FUNCTION_BLOCK "LAnyAxis_MC_OffsetRelative"   // FB30028, SCL
TITLE = LAnyAxis_MC_OffsetRelative
{ S7_Optimized_Access := 'TRUE' }
AUTHOR : tech.team.motioncontrol@siemens.com
FAMILY : AnyAxis
VERSION : 1.1
// Support: tech.team.motioncontrol@siemens.com 
// This block is for internal use only
   VAR_INPUT
      Slave : DB_ANY;   // See corresponding parameter of MC_ instruction in TIA Portal help (information system)
      Execute : Bool;   // See corresponding parameter of MC_ instruction in TIA Portal help (information system)
      Offset : LReal;   // See corresponding parameter of MC_ instruction in TIA Portal help (information system)
      ProfileReference : DInt := 1;   // See corresponding parameter of MC_ instruction in TIA Portal help (information system)
      OffsetDistance : LReal;   // See corresponding parameter of MC_ instruction in TIA Portal help (information system)
      StartPosition : LReal;   // See corresponding parameter of MC_ instruction in TIA Portal help (information system)
      Direction : DInt := 3;   // See corresponding parameter of MC_ instruction in TIA Portal help (information system)
   END_VAR
   VAR_OUTPUT
      Done : Bool;   // See corresponding parameter of MC_ instruction in TIA Portal help (information system)
      Busy : Bool;   // See corresponding parameter of MC_ instruction in TIA Portal help (information system)
      CommandAborted : Bool;   // See corresponding parameter of MC_ instruction in TIA Portal help (information system)
      Error : Bool;   // See corresponding parameter of MC_ instruction in TIA Portal help (information system)
      ErrorID : Word;   // See corresponding parameter of MC_ instruction in TIA Portal help (information system)
      CoveredOffset : LReal;   // See corresponding parameter of MC_ instruction in TIA Portal help (information system)
      StartOffset : Bool;   // See corresponding parameter of MC_ instruction in TIA Portal help (information system)
   END_VAR
   VAR CONSTANT
      ERROR_INVALID_TECHNOLOGY_OBJECT : Word := 16#8002;   // See corresponding parameter of MC_ instruction in TIA Portal help (information system)
   END_VAR
BEGIN
   REGION HEADER
     //================================================================================
     // SIEMENS AG
     // (c)Copyright 2021 All Rights Reserved
     //--------------------------------------------------------------------------------
     // Library: LAnyAxis 
     // Tested with: S7-1515-2 PN
     // Engineering: TIA Portal V17
     // Restrictions: -
     // Requirements: S7-1500 FW 2.9 
     // Functionality: Conversion DB_ANY --> TO_Axis
     // Support: tech.team.motioncontrol@siemens.com
     // Note: Parameter comments are only available in language 'English (United States)'
     //--------------------------------------------------------------------------------
     // Change log table:
     // Version  Date        Expert in charge  Changes applied
     // 01.00.00 10.03.2020  RS                First released version
     // 01.01.00 24.02.2021  RS                Update MC V6.0
     //================================================================================
   END_REGION

   #Done := FALSE;
   #Busy := FALSE;
   #CommandAborted := FALSE;
   #CoveredOffset := 0.0;
   #StartOffset := FALSE;

   IF #Execute THEN
     #Error := TRUE;
     #ErrorID := #ERROR_INVALID_TECHNOLOGY_OBJECT;
   ELSE
     #Error := FALSE;
     #ErrorID := 16#0000;
   END_IF;
END_FUNCTION_BLOCK

FUNCTION_BLOCK "LAnyAxis_MC_OffsetAbsolute"   // FB30029, SCL
TITLE = LAnyAxis_MC_OffsetAbsolute
{ S7_Optimized_Access := 'TRUE' }
AUTHOR : tech.team.motioncontrol@siemens.com
FAMILY : AnyAxis
VERSION : 1.1
// Support: tech.team.motioncontrol@siemens.com 
// This block is for internal use only
   VAR_INPUT
      Slave : DB_ANY;   // See corresponding parameter of MC_ instruction in TIA Portal help (information system)
      Execute : Bool;   // See corresponding parameter of MC_ instruction in TIA Portal help (information system)
      Offset : LReal;   // See corresponding parameter of MC_ instruction in TIA Portal help (information system)
      ProfileReference : DInt := 1;   // See corresponding parameter of MC_ instruction in TIA Portal help (information system)
      OffsetDistance : LReal;   // See corresponding parameter of MC_ instruction in TIA Portal help (information system)
      StartPosition : LReal;   // See corresponding parameter of MC_ instruction in TIA Portal help (information system)
      Direction : DInt := 3;   // See corresponding parameter of MC_ instruction in TIA Portal help (information system)
   END_VAR
   VAR_OUTPUT
      Done : Bool;   // See corresponding parameter of MC_ instruction in TIA Portal help (information system)
      Busy : Bool;   // See corresponding parameter of MC_ instruction in TIA Portal help (information system)
      CommandAborted : Bool;   // See corresponding parameter of MC_ instruction in TIA Portal help (information system)
      Error : Bool;   // See corresponding parameter of MC_ instruction in TIA Portal help (information system)
      ErrorID : Word;   // See corresponding parameter of MC_ instruction in TIA Portal help (information system)
      AbsoluteOffset : LReal;   // See corresponding parameter of MC_ instruction in TIA Portal help (information system)
      StartOffset : Bool;   // See corresponding parameter of MC_ instruction in TIA Portal help (information system)
   END_VAR
   VAR CONSTANT
      ERROR_INVALID_TECHNOLOGY_OBJECT : Word := 16#8002;   // See corresponding parameter of MC_ instruction in TIA Portal help (information system)
   END_VAR
BEGIN
   REGION HEADER
     //================================================================================
     // SIEMENS AG
     // (c)Copyright 2021 All Rights Reserved
     //--------------------------------------------------------------------------------
     // Library: LAnyAxis 
     // Tested with: S7-1515-2 PN
     // Engineering: TIA Portal V17
     // Restrictions: -
     // Requirements: S7-1500 FW 2.9 
     // Functionality: Conversion DB_ANY --> TO_Axis
     // Support: tech.team.motioncontrol@siemens.com
     // Note: Parameter comments are only available in language 'English (United States)'
     //--------------------------------------------------------------------------------
     // Change log table:
     // Version  Date        Expert in charge  Changes applied
     // 01.00.00 10.03.2020  RS                First released version
     // 01.01.00 24.02.2021  RS                Update MC V6.0
     //================================================================================
   END_REGION

   #Done := FALSE;
   #Busy := FALSE;
   #CommandAborted := FALSE;
   #AbsoluteOffset := 0.0;
   #StartOffset := FALSE;

   IF #Execute THEN
     #Error := TRUE;
     #ErrorID := #ERROR_INVALID_TECHNOLOGY_OBJECT;
   ELSE
     #Error := FALSE;
     #ErrorID := 16#0000;
   END_IF;
END_FUNCTION_BLOCK

FUNCTION_BLOCK "LAnyAxis_MC_GearOut"   // FB30032, SCL
TITLE = LAnyAxis_MC_GearOut
{ S7_Optimized_Access := 'TRUE' }
AUTHOR : tech.team.motioncontrol@siemens.com
FAMILY : AnyAxis
VERSION : 1.1
// Support: tech.team.motioncontrol@siemens.com 
// This block is for internal use only
   VAR_INPUT
      Slave : DB_ANY;   // See corresponding parameter of MC_ instruction in TIA Portal help (information system)
      Execute : Bool;   // See corresponding parameter of MC_ instruction in TIA Portal help (information system)
      SlavePosition : LReal;   // See corresponding parameter of MC_ instruction in TIA Portal help (information system)
      SyncProfileReference : DInt := 1;   // See corresponding parameter of MC_ instruction in TIA Portal help (information system)
      MasterStopDistance : LReal;   // See corresponding parameter of MC_ instruction in TIA Portal help (information system)
      Deceleration : LReal := -1.0;   // See corresponding parameter of MC_ instruction in TIA Portal help (information system)
      Jerk : LReal := -1.0;   // See corresponding parameter of MC_ instruction in TIA Portal help (information system)
      SyncOutDirection : DInt := 3;   // See corresponding parameter of MC_ instruction in TIA Portal help (information system)
   END_VAR
   VAR_OUTPUT
      StartSyncOut : Bool;   // See corresponding parameter of MC_ instruction in TIA Portal help (information system)
      Done : Bool;   // See corresponding parameter of MC_ instruction in TIA Portal help (information system)
      Busy : Bool;   // See corresponding parameter of MC_ instruction in TIA Portal help (information system)
      CommandAborted : Bool;   // See corresponding parameter of MC_ instruction in TIA Portal help (information system)
      Error : Bool;   // See corresponding parameter of MC_ instruction in TIA Portal help (information system)
      ErrorID : Word;   // See corresponding parameter of MC_ instruction in TIA Portal help (information system)
   END_VAR
   VAR CONSTANT
      ERROR_INVALID_TECHNOLOGY_OBJECT : Word := 16#8002;   // See corresponding parameter of MC_ instruction in TIA Portal help (information system)
   END_VAR
BEGIN
   REGION HEADER
     //================================================================================
     // SIEMENS AG
     // (c)Copyright 2021 All Rights Reserved
     //--------------------------------------------------------------------------------
     // Library: LAnyAxis 
     // Tested with: S7-1515-2 PN
     // Engineering: TIA Portal V17
     // Restrictions: -
     // Requirements: S7-1500 FW 2.9 
     // Functionality: Conversion DB_ANY --> TO_Axis
     // Support: tech.team.motioncontrol@siemens.com
     // Note: Parameter comments are only available in language 'English (United States)'
     //--------------------------------------------------------------------------------
     // Change log table:
     // Version  Date        Expert in charge  Changes applied
     // 01.00.00 10.03.2020  RS                First released version
     // 01.01.00 24.02.2021  RS                Update MC V6.0
     //================================================================================
   END_REGION

   #StartSyncOut := FALSE;
   #Done := FALSE;
   #Busy := FALSE;
   #CommandAborted := FALSE;

   IF #Execute THEN
     #Error := TRUE;
     #ErrorID := #ERROR_INVALID_TECHNOLOGY_OBJECT;
   ELSE
     #Error := FALSE;
     #ErrorID := 16#0000;
   END_IF;
END_FUNCTION_BLOCK

FUNCTION_BLOCK "LAnyAxis_MC_CamOut"   // FB30033, SCL
TITLE = LAnyAxis_MC_CamOut
{ S7_Optimized_Access := 'TRUE' }
AUTHOR : tech.team.motioncontrol@siemens.com
FAMILY : AnyAxis
VERSION : 1.1
// Support: tech.team.motioncontrol@siemens.com 
// This block is for internal use only
   VAR_INPUT
      Slave : DB_ANY;   // See corresponding parameter of MC_ instruction in TIA Portal help (information system)
      Execute : Bool;   // See corresponding parameter of MC_ instruction in TIA Portal help (information system)
      SlavePosition : LReal;   // See corresponding parameter of MC_ instruction in TIA Portal help (information system)
      SyncProfileReference : DInt := 1;   // See corresponding parameter of MC_ instruction in TIA Portal help (information system)
      MasterStopDistance : LReal;   // See corresponding parameter of MC_ instruction in TIA Portal help (information system)
      Deceleration : LReal := -1.0;   // See corresponding parameter of MC_ instruction in TIA Portal help (information system)
      Jerk : LReal := -1.0;   // See corresponding parameter of MC_ instruction in TIA Portal help (information system)
      SyncOutDirection : DInt := 3;   // See corresponding parameter of MC_ instruction in TIA Portal help (information system)
   END_VAR
   VAR_OUTPUT
      StartSyncOut : Bool;   // See corresponding parameter of MC_ instruction in TIA Portal help (information system)
      Done : Bool;   // See corresponding parameter of MC_ instruction in TIA Portal help (information system)
      Busy : Bool;   // See corresponding parameter of MC_ instruction in TIA Portal help (information system)
      CommandAborted : Bool;   // See corresponding parameter of MC_ instruction in TIA Portal help (information system)
      Error : Bool;   // See corresponding parameter of MC_ instruction in TIA Portal help (information system)
      ErrorID : Word;   // See corresponding parameter of MC_ instruction in TIA Portal help (information system)
   END_VAR
   VAR CONSTANT
      ERROR_INVALID_TECHNOLOGY_OBJECT : Word := 16#8002;   // See corresponding parameter of MC_ instruction in TIA Portal help (information system)
   END_VAR
BEGIN
   REGION HEADER
     //================================================================================
     // SIEMENS AG
     // (c)Copyright 2021 All Rights Reserved
     //--------------------------------------------------------------------------------
     // Library: LAnyAxis 
     // Tested with: S7-1515-2 PN
     // Engineering: TIA Portal V17
     // Restrictions: -
     // Requirements: S7-1500 FW 2.9 
     // Functionality: Conversion DB_ANY --> TO_Axis
     // Support: tech.team.motioncontrol@siemens.com
     // Note: Parameter comments are only available in language 'English (United States)'
     //--------------------------------------------------------------------------------
     // Change log table:
     // Version  Date        Expert in charge  Changes applied
     // 01.00.00 10.03.2020  RS                First released version
     // 01.01.00 24.02.2021  RS                Update MC V6.0
     //================================================================================
   END_REGION

   #StartSyncOut := FALSE;
   #Done := FALSE;
   #Busy := FALSE;
   #CommandAborted := FALSE;

   IF #Execute THEN
     #Error := TRUE;
     #ErrorID := #ERROR_INVALID_TECHNOLOGY_OBJECT;
   ELSE
     #Error := FALSE;
     #ErrorID := 16#0000;
   END_IF;
END_FUNCTION_BLOCK

// folder: LAnyAxis_Blocks/LAnyAxis_MC_SynchronousMotion/InternalSubBlocks/MC_GearIn

FUNCTION "LAnyAxis_UnpubGearInMasterExtEncoder" : Void   // FC30000, SCL
TITLE = LAnyAxis_UnpubGearInMasterExtEncoder
{ S7_Optimized_Access := 'TRUE' }
AUTHOR : tech.team.motioncontrol@siemens.com
FAMILY : AnyAxis
VERSION : 1.0
// Support: tech.team.motioncontrol@siemens.com
   VAR_INPUT
      slave : TO_SynchronousAxis;   // Slave axis specification
      master : TO_ExternalEncoder;   // Master axis specification
   END_VAR
   VAR_IN_OUT
      instMC : MC_GEARIN;   // Instance of MC_Instruction
   END_VAR
   // Ret_Val : No return value
BEGIN
   // Call of MC_Instruction
   #instMC(Master := #master,
           Slave := #slave);
END_FUNCTION

FUNCTION "LAnyAxis_UnpubGearInMasterPosAxis" : Void   // FC30001, SCL
TITLE = LAnyAxis_UnpubGearInMasterPosAxis
{ S7_Optimized_Access := 'TRUE' }
AUTHOR : tech.team.motioncontrol@siemens.com
FAMILY : AnyAxis
VERSION : 1.0
// Support: tech.team.motioncontrol@siemens.com
   VAR_INPUT
      slave : TO_SynchronousAxis;   // Slave axis specification
      master : TO_PositioningAxis;   // Master axis specification
   END_VAR
   VAR_IN_OUT
      instMC : MC_GEARIN;   // Instance of MC_Instruction
   END_VAR
   // Ret_Val : No return value
BEGIN
   // Call of MC_Instruction
   #instMC(Master := #master,
           Slave := #slave);
END_FUNCTION

FUNCTION "LAnyAxis_UnpubGearInMasterSyncAxis" : Void   // FC30002, SCL
TITLE = LAnyAxis_UnpubGearInMasterSyncAxis
{ S7_Optimized_Access := 'TRUE' }
AUTHOR : tech.team.motioncontrol@siemens.com
FAMILY : AnyAxis
VERSION : 1.0
// Support: tech.team.motioncontrol@siemens.com
   VAR_INPUT
      slave : TO_SynchronousAxis;   // Slave axis specification
      master : TO_SynchronousAxis;   // Master axis specification
   END_VAR
   VAR_IN_OUT
      instMC : MC_GEARIN;   // Instance of MC_Instruction
   END_VAR
   // Ret_Val : No return value
BEGIN
   // Call of MC_Instruction
   #instMC(Master := #master,
           Slave := #slave);
END_FUNCTION

// folder: LAnyAxis_Blocks/LAnyAxis_MC_TorqueData

FUNCTION_BLOCK "LAnyAxis_MC_TorqueLimiting"   // FB30042, SCL
TITLE = LAnyAxis_MC_TorqueLimiting
{ S7_Optimized_Access := 'TRUE' }
AUTHOR : tech.team.motioncontrol@siemens.com
FAMILY : AnyAxis
VERSION : 1.0
// Support: tech.team.motioncontrol@siemens.com 
// See corresponding MC_ instruction in TIA Portal help (information system)
   VAR_INPUT
      Axis : DB_ANY;   // See corresponding parameter of MC_ instruction in TIA Portal help (information system)
      Enable : Bool;   // See corresponding parameter of MC_ instruction in TIA Portal help (information system)
      Limit : LReal := -1.0;   // See corresponding parameter of MC_ instruction in TIA Portal help (information system)
      Mode : DInt;   // See corresponding parameter of MC_ instruction in TIA Portal help (information system)
   END_VAR
   VAR_OUTPUT
      InClamping : Bool;   // See corresponding parameter of MC_ instruction in TIA Portal help (information system)
      InLimitation : Bool;   // See corresponding parameter of MC_ instruction in TIA Portal help (information system)
      Busy : Bool;   // See corresponding parameter of MC_ instruction in TIA Portal help (information system)
      Error : Bool;   // See corresponding parameter of MC_ instruction in TIA Portal help (information system)
      ErrorId : Word;   // See corresponding parameter of MC_ instruction in TIA Portal help (information system)
   END_VAR
   VAR
      instMC : MC_TORQUELIMITING;   // Instance of MC_Instruction
      statEnableOld : Bool;   // Old value of execute
      statAxis : DB_ANY;   // Internal variable of axis
      statAxisType : Int;   // Actual state / axis type
   END_VAR
   VAR CONSTANT
      ERROR_INVALID_TECHNOLOGY_OBJECT : Word := 16#8002;   // See corresponding parameter of MC_ instruction in TIA Portal help (information system)
      IDLE : Int := 0;   // State idle
      INVALID_AXIS : Int := -1;   // Axis type: Invalid
      SPEED_AXIS : Int := 2;   // Axis type: Speed axis
      POSITIONING_AXIS : Int := 3;   // Axis type: Positioning axis
      SYNCHRONOUS_AXIS : Int := 4;   // Axis type: Synchronous axis
   END_VAR
BEGIN
   REGION HEADER
     //================================================================================
     // SIEMENS AG
     // (c)Copyright 2020 All Rights Reserved
     //--------------------------------------------------------------------------------
     // Library: LAnyAxis 
     // Tested with: S7-1515-2 PN
     // Engineering: TIA Portal V16
     // Restrictions: -
     // Requirements: S7-1500 FW 2.8.1
     // Functionality: Conversion DB_ANY --> TO_Axis
     // Support: tech.team.motioncontrol@siemens.com
     // Note: Parameter comments are only available in language 'English (United States)'
     //--------------------------------------------------------------------------------
     // Change log table:
     // Version  Date        Expert in charge  Changes applied
     // 01.00.00 10.03.2020  RS                First released version
     //================================================================================
   END_REGION

   REGION ENABLE
     IF (#statAxisType = #IDLE) AND #Enable THEN
       // Check axis type
       CASE TypeOfDB(#Axis) OF
         TO_POSITIONINGAXIS:
           #statAxisType := #POSITIONING_AXIS;
           #statAxis := #Axis;

         TO_SYNCHRONOUSAXIS:
           #statAxisType := #SYNCHRONOUS_AXIS;
           #statAxis := #Axis;

         TO_SPEEDAXIS:
           #statAxisType := #SPEED_AXIS;
           #statAxis := #Axis;

         ELSE
           #statAxisType := #INVALID_AXIS;
           #statAxis := 0;
       END_CASE;

     ELSIF NOT #Enable AND (#statAxisType = #INVALID_AXIS) THEN
       #statAxisType := #IDLE;

       // Outputs
       #InClamping := FALSE;
       #InLimitation := FALSE;
       #Busy := FALSE;
       #Error := FALSE;
       #ErrorId := 16#0;
     END_IF;

     // Edge detection
     #statEnableOld := #Enable;
   END_REGION

   CASE #statAxisType OF
     #IDLE:
       ;

     #POSITIONING_AXIS,
     #SYNCHRONOUS_AXIS,
     #SPEED_AXIS:
       REGION VALID_AXIS
         // Inputs
         #instMC.Enable := #Enable;
         #instMC.Limit := #Limit;
         #instMC.Mode := #Mode;

         // Call of MC instruction
         CASE #statAxisType OF
           #POSITIONING_AXIS:
             "LAnyAxis_UnpubTorqueLimitingPosAxis"(axis := #statAxis,
                                                   instMC := #instMC);
           #SYNCHRONOUS_AXIS:
             "LAnyAxis_UnpubTorqueLimitingSyncAxis"(axis := #statAxis,
                                                    instMC := #instMC);
           #SPEED_AXIS:
             #instMC(Axis := #statAxis);
         END_CASE;

         // Outputs
         #InClamping := #instMC.InClamping;
         #InLimitation := #instMC.InLimitation;
         #Busy := #instMC.Busy;
         #Error := #instMC.Error;
         #ErrorId := #instMC.ErrorId;

         // Status of MC instruction
         IF NOT #instMC.Busy
           AND NOT #instMC.Error
         THEN
           // Not active
           #statAxisType := #IDLE;
         END_IF;
       END_REGION

     ELSE
       REGION INVALID_AXIS
         // Outputs
         #InClamping := FALSE;
         #InLimitation := FALSE;
         #Busy := FALSE;
         #Error := TRUE;
         #ErrorId := #ERROR_INVALID_TECHNOLOGY_OBJECT;
       END_REGION
   END_CASE;
END_FUNCTION_BLOCK

// folder: LAnyAxis_Blocks/LAnyAxis_MC_TorqueData/InternalSubBlocks/MC_TorqueLimiting

FUNCTION "LAnyAxis_UnpubTorqueLimitingPosAxis" : Void   // FC30032, SCL
TITLE = LAnyAxis_UnpubTorqueLimitingPosAxis
{ S7_Optimized_Access := 'TRUE' }
AUTHOR : tech.team.motioncontrol@siemens.com
FAMILY : AnyAxis
VERSION : 1.0
// Support: tech.team.motioncontrol@siemens.com
   VAR_INPUT
      axis : TO_PositioningAxis;   // Axis specification
   END_VAR
   VAR_IN_OUT
      instMC : MC_TORQUELIMITING;   // Instance of MC_Instruction
   END_VAR
   // Ret_Val : No return value
BEGIN
   // Call of MC_Instruction
   #instMC(Axis := #axis);
END_FUNCTION

FUNCTION "LAnyAxis_UnpubTorqueLimitingSyncAxis" : Void   // FC30034, SCL
TITLE = LAnyAxis_UnpubTorqueLimitingSyncAxis
{ S7_Optimized_Access := 'TRUE' }
AUTHOR : tech.team.motioncontrol@siemens.com
FAMILY : AnyAxis
VERSION : 1.0
// Support: tech.team.motioncontrol@siemens.com
   VAR_INPUT
      axis : TO_SynchronousAxis;   // Axis specification
   END_VAR
   VAR_IN_OUT
      instMC : MC_TORQUELIMITING;   // Instance of MC_Instruction
   END_VAR
   // Ret_Val : No return value
BEGIN
   // Call of MC_Instruction
   #instMC(Axis := #axis);
END_FUNCTION

// folder: LAnyAxis_Blocks/LAnyAxis_TagsAccess

FUNCTION "LAnyAxis_StatusWord" : Word   // FC30077, SCL
TITLE = LAnyAxis_StatusWord
{ S7_Optimized_Access := 'TRUE' }
AUTHOR : tech.team.motioncontrol@siemens.com
FAMILY : AnyAxis
VERSION : 1.0
// Support: tech.team.motioncontrol@siemens.com
   VAR_INPUT
      axis : DB_ANY;   // Axis specification
   END_VAR
   VAR_OUTPUT
      statusWord : DWord;   // axis.StatusWord
   END_VAR
   // Ret_Val : Return value
   VAR CONSTANT
      ERROR_INVALID_TECHNOLOGY_OBJECT : Word := 16#8002;   // Error invalid TO specification
      FINISHED : Word := 16#0000;   // Finished without error
   END_VAR
BEGIN
   REGION HEADER
     //================================================================================
     // SIEMENS AG
     // (c)Copyright 2020 All Rights Reserved
     //--------------------------------------------------------------------------------
     // Library: LAnyAxis 
     // Tested with: S7-1515-2 PN
     // Engineering: TIA Portal V16
     // Restrictions: -
     // Requirements: S7-1500 FW 2.8.1
     // Functionality: Conversion DB_ANY --> TO_Axis
     // Support: tech.team.motioncontrol@siemens.com
     // Note: Parameter comments are only available in language 'English (United States)'
     //--------------------------------------------------------------------------------
     // Change log table:
     // Version  Date        Expert in charge  Changes applied
     // 01.00.00 10.03.2020  RS                First released version
     //================================================================================
   END_REGION

   // Read axis parameter
   CASE TypeOfDB(#axis) OF
     TO_POSITIONINGAXIS:
       #statusWord := "LAnyAxis_UnpubStatusWordPosAxis"(#axis);
       #LAnyAxis_StatusWord := #FINISHED;

     TO_SYNCHRONOUSAXIS:
       #statusWord := "LAnyAxis_UnpubStatusWordSyncAxis"(#axis);
       #LAnyAxis_StatusWord := #FINISHED;

     TO_EXTERNALENCODER:
       #statusWord := "LAnyAxis_UnpubStatusWordExtEncoder"(#axis);
       #LAnyAxis_StatusWord := #FINISHED;

     TO_SPEEDAXIS:
       #statusWord := "LAnyAxis_UnpubStatusWordSpeedAxis"(#axis);
       #LAnyAxis_StatusWord := #FINISHED;

     ELSE
       #LAnyAxis_StatusWord := #ERROR_INVALID_TECHNOLOGY_OBJECT; // Invalid TO specification
   END_CASE;
END_FUNCTION

FUNCTION "LAnyAxis_StatusWord2" : Word   // FC30081, SCL
TITLE = LAnyAxis_StatusWord2
{ S7_Optimized_Access := 'TRUE' }
AUTHOR : tech.team.motioncontrol@siemens.com
FAMILY : AnyAxis
VERSION : 1.0
// Support: tech.team.motioncontrol@siemens.com
   VAR_INPUT
      axis : DB_ANY;   // Axis specification
   END_VAR
   VAR_OUTPUT
      statusWord2 : DWord;   // axis.StatusWord2
   END_VAR
   // Ret_Val : Return value
   VAR CONSTANT
      ERROR_INVALID_TECHNOLOGY_OBJECT : Word := 16#8002;   // Error invalid TO specification
      FINISHED : Word := 16#0000;   // Finished without error
   END_VAR
BEGIN
   REGION HEADER
     //================================================================================
     // SIEMENS AG
     // (c)Copyright 2020 All Rights Reserved
     //--------------------------------------------------------------------------------
     // Library: LAnyAxis 
     // Tested with: S7-1515-2 PN
     // Engineering: TIA Portal V16
     // Restrictions: -
     // Requirements: S7-1500 FW 2.8.1
     // Functionality: Conversion DB_ANY --> TO_Axis
     // Support: tech.team.motioncontrol@siemens.com
     // Note: Parameter comments are only available in language 'English (United States)'
     //--------------------------------------------------------------------------------
     // Change log table:
     // Version  Date        Expert in charge  Changes applied
     // 01.00.00 10.03.2020  RS                First released version
     //================================================================================
   END_REGION

   // Read axis parameter
   CASE TypeOfDB(#axis) OF
     TO_POSITIONINGAXIS:
       #statusWord2 := "LAnyAxis_UnpubStatusWord2PosAxis"(#axis);
       #LAnyAxis_StatusWord2 := #FINISHED;

     TO_SYNCHRONOUSAXIS:
       #statusWord2 := "LAnyAxis_UnpubStatusWord2SyncAxis"(#axis);
       #LAnyAxis_StatusWord2 := #FINISHED;

     TO_SPEEDAXIS:
       #statusWord2 := "LAnyAxis_UnpubStatusWord2SpeedAxis"(#axis);
       #LAnyAxis_StatusWord2 := #FINISHED;

     ELSE
       #LAnyAxis_StatusWord2 := #ERROR_INVALID_TECHNOLOGY_OBJECT; // Invalid TO specification
   END_CASE;
END_FUNCTION

FUNCTION "LAnyAxis_Position" : Word   // FC30087, SCL
TITLE = LAnyAxis_Position
{ S7_Optimized_Access := 'TRUE' }
AUTHOR : tech.team.motioncontrol@siemens.com
FAMILY : AnyAxis
VERSION : 1.1
// Support: tech.team.motioncontrol@siemens.com
   VAR_INPUT
      axis : DB_ANY;   // Axis specification
   END_VAR
   VAR_OUTPUT
      position : LReal;   // axis.Position
   END_VAR
   // Ret_Val : Return value
   VAR CONSTANT
      ERROR_INVALID_TECHNOLOGY_OBJECT : Word := 16#8002;   // Error invalid TO specification
      FINISHED : Word := 16#0000;   // Finished without error
   END_VAR
BEGIN
   REGION HEADER
     //================================================================================
     // SIEMENS AG
     // (c)Copyright 2021 All Rights Reserved
     //--------------------------------------------------------------------------------
     // Library: LAnyAxis 
     // Tested with: S7-1515-2 PN
     // Engineering: TIA Portal V17
     // Restrictions: -
     // Requirements: S7-1500 FW 2.9
     // Functionality: Conversion DB_ANY --> TO_Axis
     // Support: tech.team.motioncontrol@siemens.com
     // Note: Parameter comments are only available in language 'English (United States)'
     //--------------------------------------------------------------------------------
     // Change log table:
     // Version  Date        Expert in charge  Changes applied
     // 01.00.00 01.01.2021  RS                First released version
     // 01.01.00 24.02.2021  RS                Update MC V6.0
     //================================================================================
   END_REGION

   // Read axis parameter
   CASE TypeOfDB(#axis) OF
     TO_POSITIONINGAXIS:
       #position := "LAnyAxis_UnpubPositionPosAxis"(#axis);
       #LAnyAxis_Position := #FINISHED;

     TO_SYNCHRONOUSAXIS:
       #position := "LAnyAxis_UnpubPositionSyncAxis"(#axis);
       #LAnyAxis_Position := #FINISHED;

     ELSE
       #LAnyAxis_Position := #ERROR_INVALID_TECHNOLOGY_OBJECT; // Invalid TO specification
   END_CASE;
END_FUNCTION

// folder: LAnyAxis_Blocks/LAnyAxis_TagsAccess/InternalSubBlocks/Position

FUNCTION "LAnyAxis_UnpubPositionPosAxis" : LReal   // FC30085, SCL
TITLE = LAnyAxis_UnpubPositionPosAxis
{ S7_Optimized_Access := 'TRUE' }
AUTHOR : tech.team.motioncontrol@siemens.com
FAMILY : AnyAxis
VERSION : 1.0
// Support: tech.team.motioncontrol@siemens.com
   VAR_INPUT
      axis : TO_PositioningAxis;   // Axis specification
   END_VAR
   // Ret_Val : axis.Position
BEGIN
   // Read axis parameter
   #LAnyAxis_UnpubPositionPosAxis := #axis.Position;
END_FUNCTION

FUNCTION "LAnyAxis_UnpubPositionSyncAxis" : LReal   // FC30086, SCL
TITLE = LAnyAxis_UnpubPositionSyncAxis
{ S7_Optimized_Access := 'TRUE' }
AUTHOR : tech.team.motioncontrol@siemens.com
FAMILY : AnyAxis
VERSION : 1.0
// Support: tech.team.motioncontrol@siemens.com
   VAR_INPUT
      axis : TO_SynchronousAxis;   // Axis specification
   END_VAR
   // Ret_Val : axis.Position
BEGIN
   // Read axis parameter
   #LAnyAxis_UnpubPositionSyncAxis := #axis.Position;
END_FUNCTION

// folder: LAnyAxis_Blocks/LAnyAxis_TagsAccess/InternalSubBlocks/StatusWord

FUNCTION "LAnyAxis_UnpubStatusWordExtEncoder" : DWord   // FC30073, SCL
TITLE = LAnyAxis_UnpubStatusWordExtEncoder
{ S7_Optimized_Access := 'TRUE' }
AUTHOR : tech.team.motioncontrol@siemens.com
FAMILY : AnyAxis
VERSION : 1.0
// Support: tech.team.motioncontrol@siemens.com
   VAR_INPUT
      axis : TO_ExternalEncoder;   // Axis specification
   END_VAR
   // Ret_Val : axis.StatusWord
BEGIN
   // Read axis parameter
   #LAnyAxis_UnpubStatusWordExtEncoder := #axis.StatusWord;
END_FUNCTION

FUNCTION "LAnyAxis_UnpubStatusWordPosAxis" : DWord   // FC30074, SCL
TITLE = LAnyAxis_UnpubStatusWordPosAxis
{ S7_Optimized_Access := 'TRUE' }
AUTHOR : tech.team.motioncontrol@siemens.com
FAMILY : AnyAxis
VERSION : 1.0
// Support: tech.team.motioncontrol@siemens.com
   VAR_INPUT
      axis : TO_PositioningAxis;   // Axis specification
   END_VAR
   // Ret_Val : axis.StatusWord
BEGIN
   // Read axis parameter
   #LAnyAxis_UnpubStatusWordPosAxis := #axis.StatusWord;
END_FUNCTION

FUNCTION "LAnyAxis_UnpubStatusWordSyncAxis" : DWord   // FC30076, SCL
TITLE = LAnyAxis_UnpubStatusWordSyncAxis
{ S7_Optimized_Access := 'TRUE' }
AUTHOR : tech.team.motioncontrol@siemens.com
FAMILY : AnyAxis
VERSION : 1.0
// Support: tech.team.motioncontrol@siemens.com
   VAR_INPUT
      axis : TO_SynchronousAxis;   // Axis specification
   END_VAR
   // Ret_Val : axis.StatusWord
BEGIN
   // Read axis parameter
   #LAnyAxis_UnpubStatusWordSyncAxis := #axis.StatusWord;
END_FUNCTION

FUNCTION "LAnyAxis_UnpubStatusWordSpeedAxis" : DWord   // FC30079, SCL
TITLE = LAnyAxis_UnpubStatusWordSpeedAxis
{ S7_Optimized_Access := 'TRUE' }
AUTHOR : tech.team.motioncontrol@siemens.com
FAMILY : AnyAxis
VERSION : 1.0
// Support: tech.team.motioncontrol@siemens.com
   VAR_INPUT
      axis : TO_SpeedAxis;   // Axis specification
   END_VAR
   // Ret_Val : axis.StatusWord
BEGIN
   // Read axis parameter
   #LAnyAxis_UnpubStatusWordSpeedAxis := #axis.StatusWord;
END_FUNCTION

// folder: LAnyAxis_Blocks/LAnyAxis_TagsAccess/InternalSubBlocks/StatusWord2

FUNCTION "LAnyAxis_UnpubStatusWord2SpeedAxis" : DWord   // FC30072, SCL
TITLE = LAnyAxis_UnpubStatusWordSpeedAxis
{ S7_Optimized_Access := 'TRUE' }
AUTHOR : tech.team.motioncontrol@siemens.com
FAMILY : AnyAxis
VERSION : 1.0
// Support: tech.team.motioncontrol@siemens.com
   VAR_INPUT
      axis : TO_SpeedAxis;   // Axis specification
   END_VAR
   // Ret_Val : axis.StatusWord2
BEGIN
   // Read axis parameter
   #LAnyAxis_UnpubStatusWord2SpeedAxis := #axis.StatusWord2;
END_FUNCTION

FUNCTION "LAnyAxis_UnpubStatusWord2PosAxis" : DWord   // FC30078, SCL
TITLE = LAnyAxis_UnpubStatusWord2PosAxis
{ S7_Optimized_Access := 'TRUE' }
AUTHOR : tech.team.motioncontrol@siemens.com
FAMILY : AnyAxis
VERSION : 1.0
// Support: tech.team.motioncontrol@siemens.com
   VAR_INPUT
      axis : TO_PositioningAxis;   // Axis specification
   END_VAR
   // Ret_Val : axis.StatusWord2
BEGIN
   // Read axis parameter
   #LAnyAxis_UnpubStatusWord2PosAxis := #axis.StatusWord2;
END_FUNCTION

FUNCTION "LAnyAxis_UnpubStatusWord2SyncAxis" : DWord   // FC30080, SCL
TITLE = LAnyAxis_UnpubStatusWord2SyncAxis
{ S7_Optimized_Access := 'TRUE' }
AUTHOR : tech.team.motioncontrol@siemens.com
FAMILY : AnyAxis
VERSION : 1.0
// Support: tech.team.motioncontrol@siemens.com
   VAR_INPUT
      axis : TO_SynchronousAxis;   // Axis specification
   END_VAR
   // Ret_Val : axis.StatusWord2
BEGIN
   // Read axis parameter
   #LAnyAxis_UnpubStatusWord2SyncAxis := #axis.StatusWord2;
END_FUNCTION

// folder: LAnyAxis_Blocks/LAnyAxis_TagsAccess/Modulo

FUNCTION "LAnyAxis_ModuloEnable" : Word   // FC30114, SCL
TITLE = LAnyAxis_ModuloEnable
{ S7_Optimized_Access := 'TRUE' }
AUTHOR : tech.team.motioncontrol@siemens.com
FAMILY : AnyAxis
VERSION : 1.1
// Support: tech.team.motioncontrol@siemens.com
   VAR_INPUT
      axis : DB_ANY;   // Axis specification
   END_VAR
   VAR_OUTPUT
      enable : Bool;   // axis.Modulo.Enable
   END_VAR
   // Ret_Val : Return value
   VAR CONSTANT
      ERROR_INVALID_TECHNOLOGY_OBJECT : Word := 16#8002;   // Error invalid TO specification
      FINISHED : Word := 16#0000;   // Finished without error
   END_VAR
BEGIN
   REGION HEADER
     //================================================================================
     // SIEMENS AG
     // (c)Copyright 2021 All Rights Reserved
     //--------------------------------------------------------------------------------
     // Library: LAnyAxis 
     // Tested with: S7-1515-2 PN
     // Engineering: TIA Portal V17
     // Restrictions: -
     // Requirements: S7-1500 FW 2.9
     // Functionality: Conversion DB_ANY --> TO_Axis
     // Support: tech.team.motioncontrol@siemens.com
     // Note: Parameter comments are only available in language 'English (United States)'
     //--------------------------------------------------------------------------------
     // Change log table:
     // Version  Date        Expert in charge  Changes applied
     // 01.00.00 01.01.2021  RS                First released version
     // 01.01.00 24.02.2021  RS                Update MC V6.0
     //================================================================================
   END_REGION

   // Read axis parameter
   CASE TypeOfDB(#axis) OF
     TO_POSITIONINGAXIS:
       #enable := "LAnyAxis_UnpubModuloEnablePosAxis"(#axis);
       #LAnyAxis_ModuloEnable := #FINISHED;

     TO_SYNCHRONOUSAXIS:
       #enable := "LAnyAxis_UnpubModuloEnableSyncAxis"(#axis);
       #LAnyAxis_ModuloEnable := #FINISHED;

     TO_EXTERNALENCODER:
       #enable := "LAnyAxis_UnpubModuloEnableExtEncoder"(#axis);
       #LAnyAxis_ModuloEnable := #FINISHED;

     ELSE
       #LAnyAxis_ModuloEnable := #ERROR_INVALID_TECHNOLOGY_OBJECT; // Invalid TO specification
   END_CASE;
END_FUNCTION

// folder: LAnyAxis_Blocks/LAnyAxis_TagsAccess/Modulo/InternalSubBlocks/Enable

FUNCTION "LAnyAxis_UnpubModuloEnableExtEncoder" : Bool   // FC30093, SCL
TITLE = LAnyAxis_UnpubModuloEnableExtEncoder
{ S7_Optimized_Access := 'TRUE' }
AUTHOR : tech.team.motioncontrol@siemens.com
FAMILY : AnyAxis
VERSION : 1.0
// Support: tech.team.motioncontrol@siemens.com
   VAR_INPUT
      axis : TO_ExternalEncoder;   // Axis specification
   END_VAR
   // Ret_Val : axis.Modulo.Enable
BEGIN
   // Read axis parameter
   #LAnyAxis_UnpubModuloEnableExtEncoder := #axis.Modulo.Enable;
END_FUNCTION

FUNCTION "LAnyAxis_UnpubModuloEnablePosAxis" : Bool   // FC30094, SCL
TITLE = LAnyAxis_UnpubModuloEnablePosAxis
{ S7_Optimized_Access := 'TRUE' }
AUTHOR : tech.team.motioncontrol@siemens.com
FAMILY : AnyAxis
VERSION : 1.0
// Support: tech.team.motioncontrol@siemens.com
   VAR_INPUT
      axis : TO_PositioningAxis;   // Axis specification
   END_VAR
   // Ret_Val : axis.Modulo.Enable
BEGIN
   // Read axis parameter
   #LAnyAxis_UnpubModuloEnablePosAxis := #axis.Modulo.Enable;
END_FUNCTION

FUNCTION "LAnyAxis_UnpubModuloEnableSyncAxis" : Bool   // FC30095, SCL
TITLE = LAnyAxis_UnpubModuloEnableSyncAxis
{ S7_Optimized_Access := 'TRUE' }
AUTHOR : tech.team.motioncontrol@siemens.com
FAMILY : AnyAxis
VERSION : 1.0
// Support: tech.team.motioncontrol@siemens.com
   VAR_INPUT
      axis : TO_SynchronousAxis;   // Axis specification
   END_VAR
   // Ret_Val : axis.Modulo.Enable
BEGIN
   // Read axis parameter
   #LAnyAxis_UnpubModuloEnableSyncAxis := #axis.Modulo.Enable;
END_FUNCTION

// ===== library: MasterCopy "S7-1500T_LAnyAxis_Blocks (Drop in folder "Program blocks")" =====

// folder: LAnyAxis_Blocks

FUNCTION_BLOCK "LAnyAxis_MC_Power"   // FB30000, SCL
TITLE = LAnyAxis_MC_Power
{ S7_Optimized_Access := 'TRUE' }
AUTHOR : tech.team.motioncontrol@siemens.com
FAMILY : AnyAxis
VERSION : 1.0
// Support: tech.team.motioncontrol@siemens.com 
// See corresponding MC_ instruction in TIA Portal help (information system)
   VAR_INPUT
      Axis : DB_ANY;   // See corresponding parameter of MC_ instruction in TIA Portal help (information system)
      Enable : Bool;   // See corresponding parameter of MC_ instruction in TIA Portal help (information system)
      StartMode : DInt := 1;   // See corresponding parameter of MC_ instruction in TIA Portal help (information system)
      StopMode : Int;   // See corresponding parameter of MC_ instruction in TIA Portal help (information system)
   END_VAR
   VAR_OUTPUT
      Status : Bool;   // See corresponding parameter of MC_ instruction in TIA Portal help (information system)
      Busy : Bool;   // See corresponding parameter of MC_ instruction in TIA Portal help (information system)
      Error : Bool;   // See corresponding parameter of MC_ instruction in TIA Portal help (information system)
      ErrorID : Word;   // See corresponding parameter of MC_ instruction in TIA Portal help (information system)
   END_VAR
   VAR
      instMC : MC_POWER;   // Instance of MC_Instruction
      statAxis : DB_ANY;   // Internal variable of axis
      statAxisType : Int;   // Actual state / axis type
   END_VAR
   VAR CONSTANT
      ERROR_INVALID_TECHNOLOGY_OBJECT : Word := 16#8002;   // See corresponding parameter of MC_ instruction in TIA Portal help (information system)
      IDLE : Int := 0;   // State idle
      INVALID_AXIS : Int := -1;   // Axis type: Invalid
      EXTERNAL_ENCODER : Int := 1;   // Axis type: External encoder
      SPEED_AXIS : Int := 2;   // Axis type: Speed axis
      POSITIONING_AXIS : Int := 3;   // Axis type: Positioning axis
      SYNCHRONOUS_AXIS : Int := 4;   // Axis type: Synchronous axis
   END_VAR
BEGIN
   REGION HEADER
     //================================================================================
     // SIEMENS AG
     // (c)Copyright 2020 All Rights Reserved
     //--------------------------------------------------------------------------------
     // Library: LAnyAxis 
     // Tested with: S7-1515-2 PN
     // Engineering: TIA Portal V16
     // Restrictions: -
     // Requirements: S7-1500 FW 2.8.1
     // Functionality: Conversion DB_ANY --> TO_Axis
     // Support: tech.team.motioncontrol@siemens.com
     // Note: Parameter comments are only available in language 'English (United States)'
     //--------------------------------------------------------------------------------
     // Change log table:
     // Version  Date        Expert in charge  Changes applied
     // 01.00.00 10.03.2020  RS                First released version
     //================================================================================
   END_REGION

   REGION ENABLE
     IF (#statAxisType = #IDLE) AND #Enable THEN
       // Check axis type
       CASE TypeOfDB(#Axis) OF
         TO_POSITIONINGAXIS:
           #statAxisType := #POSITIONING_AXIS;
           #statAxis := #Axis;

         TO_SYNCHRONOUSAXIS:
           #statAxisType := #SYNCHRONOUS_AXIS;
           #statAxis := #Axis;

         TO_SPEEDAXIS:
           #statAxisType := #SPEED_AXIS;
           #statAxis := #Axis;

         TO_EXTERNALENCODER:
           #statAxisType := #EXTERNAL_ENCODER;
           #statAxis := #Axis;
         ELSE
           #statAxisType := #INVALID_AXIS;
           #statAxis := 0;
       END_CASE;

     ELSIF NOT #Enable AND (#statAxisType = #INVALID_AXIS) THEN
       #statAxisType := #IDLE;

       // Outputs
       #Status := FALSE;
       #Busy := FALSE;
       #Error := FALSE;
       #ErrorID := 16#0000;
     END_IF;
   END_REGION

   CASE #statAxisType OF
     #IDLE:
       ;

     #POSITIONING_AXIS,
     #SYNCHRONOUS_AXIS,
     #SPEED_AXIS,
     #EXTERNAL_ENCODER:
       REGION VALID_AXIS
         // Inputs
         #instMC.Enable := #Enable;
         #instMC.StartMode := #StartMode;
         #instMC.StopMode := #StopMode;

         // Call of MC instruction
         CASE #statAxisType OF
           #POSITIONING_AXIS:
             "LAnyAxis_UnpubPowerPosAxis"(axis := #statAxis,
                                          instMC := #instMC);
           #SYNCHRONOUS_AXIS:
             "LAnyAxis_UnpubPowerSyncAxis"(axis := #statAxis,
                                           instMC := #instMC);
           #SPEED_AXIS:
             "LAnyAxis_UnpubPowerSpeedAxis"(axis := #statAxis,
                                            instMC := #instMC);
           #EXTERNAL_ENCODER:
             "LAnyAxis_UnpubPowerExtEncoder"(axis := #statAxis,
                                             instMC := #instMC);
         END_CASE;

         // Outputs
         #Status := #instMC.Status;
         #Busy := #instMC.Busy;
         #Error := #instMC.Error;
         #ErrorID := #instMC.ErrorId;

         // Status of MC instruction
         IF NOT #instMC.Busy
           AND NOT #instMC.Error
           AND NOT #instMC.Status
         THEN
           // Not active
           #statAxisType := #IDLE;
         END_IF;
       END_REGION

     ELSE
       REGION INVALID_AXIS
         // Outputs
         #Status := FALSE;
         #Busy := FALSE;
         #Error := TRUE;
         #ErrorID := #ERROR_INVALID_TECHNOLOGY_OBJECT;
       END_REGION
   END_CASE;
END_FUNCTION_BLOCK

FUNCTION_BLOCK "LAnyAxis_MC_Reset"   // FB30001, SCL
TITLE = LAnyAxis_MC_Reset
{ S7_Optimized_Access := 'TRUE' }
AUTHOR : tech.team.motioncontrol@siemens.com
FAMILY : AnyAxis
VERSION : 1.0
// Support: tech.team.motioncontrol@siemens.com 
// See corresponding MC_ instruction in TIA Portal help (information system)
   VAR_INPUT
      Axis : DB_ANY;   // See corresponding parameter of MC_ instruction in TIA Portal help (information system)
      Execute : Bool;   // See corresponding parameter of MC_ instruction in TIA Portal help (information system)
      Restart : Bool;   // See corresponding parameter of MC_ instruction in TIA Portal help (information system)
   END_VAR
   VAR_OUTPUT
      Done : Bool;   // See corresponding parameter of MC_ instruction in TIA Portal help (information system)
      Busy : Bool;   // See corresponding parameter of MC_ instruction in TIA Portal help (information system)
      CommandAborted : Bool;   // See corresponding parameter of MC_ instruction in TIA Portal help (information system)
      Error : Bool;   // See corresponding parameter of MC_ instruction in TIA Portal help (information system)
      ErrorID : Word;   // See corresponding parameter of MC_ instruction in TIA Portal help (information system)
   END_VAR
   VAR
      instMC : MC_RESET;   // Instance of MC_Instruction
      statExecuteOld : Bool;   // Old value of execute
      statAxis : DB_ANY;   // Internal variable of axis
      statAxisType : Int;   // Actual state / axis type
   END_VAR
   VAR CONSTANT
      ERROR_INVALID_TECHNOLOGY_OBJECT : Word := 16#8002;   // See corresponding parameter of MC_ instruction in TIA Portal help (information system)
      IDLE : Int := 0;   // State idle
      INVALID_AXIS : Int := -1;   // Axis type: Invalid
      EXTERNAL_ENCODER : Int := 1;   // Axis type: External encoder
      SPEED_AXIS : Int := 2;   // Axis type: Speed axis
      POSITIONING_AXIS : Int := 3;   // Axis type: Positioning axis
      SYNCHRONOUS_AXIS : Int := 4;   // Axis type: Synchronous axis
      PROXY : Int := 5;   // Axis type: Leading axis proxy
   END_VAR
BEGIN
   REGION HEADER
     //================================================================================
     // SIEMENS AG
     // (c)Copyright 2020 All Rights Reserved
     //--------------------------------------------------------------------------------
     // Library: LAnyAxis 
     // Tested with: S7-1515T-2 PN
     // Engineering: TIA Portal V16
     // Restrictions: -
     // Requirements: S7-1500T FW 2.8.1
     // Functionality: Conversion DB_ANY --> TO_Axis
     // Support: tech.team.motioncontrol@siemens.com
     // Note: Parameter comments are only available in language 'English (United States)'
     //--------------------------------------------------------------------------------
     // Change log table:
     // Version  Date        Expert in charge  Changes applied
     // 01.00.00 10.03.2020  RS                First released version
     //================================================================================
   END_REGION

   REGION EXECUTE
     IF #Execute AND NOT #statExecuteOld THEN
       // Copy parameter
       #instMC.Restart := #Restart;

       // Check axis type
       CASE TypeOfDB(#Axis) OF
         TO_POSITIONINGAXIS:
           #statAxisType := #POSITIONING_AXIS;
           #statAxis := #Axis;

         TO_SYNCHRONOUSAXIS:
           #statAxisType := #SYNCHRONOUS_AXIS;
           #statAxis := #Axis;

         TO_EXTERNALENCODER:
           #statAxisType := #EXTERNAL_ENCODER;
           #statAxis := #Axis;

         TO_SPEEDAXIS:
           #statAxisType := #SPEED_AXIS;
           #statAxis := #Axis;

         TO_LEADINGAXISPROXY:
           #statAxisType := #PROXY;
           #statAxis := #Axis;

         ELSE
           #statAxisType := #INVALID_AXIS;
           #statAxis := 0;
       END_CASE;

     ELSIF NOT #Execute AND (#statAxisType = #INVALID_AXIS) THEN
       #statAxisType := #IDLE;

       // Outputs
       #Done := FALSE;
       #Busy := FALSE;
       #CommandAborted := FALSE;
       #Error := FALSE;
       #ErrorID := 16#0000;
     END_IF;

     // Edge detection
     #statExecuteOld := #Execute;
   END_REGION

   CASE #statAxisType OF
     #IDLE:
       ;

     #POSITIONING_AXIS,
     #SYNCHRONOUS_AXIS,
     #SPEED_AXIS,
     #EXTERNAL_ENCODER,
     #PROXY:
       REGION VALID_AXIS
         // Inputs
         #instMC.Execute := #Execute;

         // Call of MC instruction
         CASE #statAxisType OF
           #POSITIONING_AXIS:
             "LAnyAxis_UnpubResetPosAxis"(axis := #statAxis,
                                          instMC := #instMC);
           #SYNCHRONOUS_AXIS:
             "LAnyAxis_UnpubResetSyncAxis"(axis := #statAxis,
                                           instMC := #instMC);
           #SPEED_AXIS:
             "LAnyAxis_UnpubResetSpeedAxis"(axis := #statAxis,
                                            instMC := #instMC);
           #EXTERNAL_ENCODER:
             "LAnyAxis_UnpubResetExtEncoder"(axis := #statAxis,
                                             instMC := #instMC);
           #PROXY:
             "LAnyAxis_UnpubResetProxy"(axis := #statAxis,
                                        instMC := #instMC);
         END_CASE;

         // Outputs
         #Done := #instMC.Done;
         #Busy := #instMC.Busy;
         #CommandAborted := #instMC.CommandAborted;
         #Error := #instMC.Error;
         #ErrorID := #instMC.ErrorId;

         // Status of MC instruction
         IF NOT #instMC.Done
           AND NOT #instMC.Busy
           AND NOT #instMC.CommandAborted
           AND NOT #instMC.Error
         THEN
           // Not active
           #statAxisType := #IDLE;
         END_IF;
       END_REGION

     ELSE
       REGION INVALID_AXIS
         // Outputs
         #Done := FALSE;
         #Busy := FALSE;
         #CommandAborted := FALSE;
         #Error := TRUE;
         #ErrorID := #ERROR_INVALID_TECHNOLOGY_OBJECT;
       END_REGION
   END_CASE;
END_FUNCTION_BLOCK

FUNCTION_BLOCK "LAnyAxis_MC_Home"   // FB30002, SCL
TITLE = LAnyAxis_MC_Home
{ S7_Optimized_Access := 'TRUE' }
AUTHOR : tech.team.motioncontrol@siemens.com
FAMILY : AnyAxis
VERSION : 1.0
// Support: tech.team.motioncontrol@siemens.com 
// See corresponding MC_ instruction in TIA Portal help (information system)
   VAR_INPUT
      Axis : DB_ANY;   // See corresponding parameter of MC_ instruction in TIA Portal help (information system)
      Execute : Bool;   // See corresponding parameter of MC_ instruction in TIA Portal help (information system)
      Position : LReal;   // See corresponding parameter of MC_ instruction in TIA Portal help (information system)
      Mode : Int;   // See corresponding parameter of MC_ instruction in TIA Portal help (information system)
   END_VAR
   VAR_OUTPUT
      ReferenceMarkPosition : LReal;   // See corresponding parameter of MC_ instruction in TIA Portal help (information system)
      Done : Bool;   // See corresponding parameter of MC_ instruction in TIA Portal help (information system)
      Busy : Bool;   // See corresponding parameter of MC_ instruction in TIA Portal help (information system)
      CommandAborted : Bool;   // See corresponding parameter of MC_ instruction in TIA Portal help (information system)
      Error : Bool;   // See corresponding parameter of MC_ instruction in TIA Portal help (information system)
      ErrorID : Word;   // See corresponding parameter of MC_ instruction in TIA Portal help (information system)
   END_VAR
   VAR
      instMC : MC_HOME;   // Instance of MC_Instruction
      statExecuteOld : Bool;   // Old value of execute
      statAxis : DB_ANY;   // Internal variable of axis
      statAxisType : Int;   // Actual state / axis type
   END_VAR
   VAR CONSTANT
      ERROR_INVALID_TECHNOLOGY_OBJECT : Word := 16#8002;   // See corresponding parameter of MC_ instruction in TIA Portal help (information system)
      IDLE : Int := 0;   // State idle
      INVALID_AXIS : Int := -1;   // Axis type: Invalid
      EXTERNAL_ENCODER : Int := 1;   // Axis type: External encoder
      POSITIONING_AXIS : Int := 3;   // Axis type: Positioning axis
      SYNCHRONOUS_AXIS : Int := 4;   // Axis type: Synchronous axis
   END_VAR
BEGIN
   REGION HEADER
     //================================================================================
     // SIEMENS AG
     // (c)Copyright 2020 All Rights Reserved
     //--------------------------------------------------------------------------------
     // Library: LAnyAxis 
     // Tested with: S7-1515-2 PN
     // Engineering: TIA Portal V16
     // Restrictions: -
     // Requirements: S7-1500 FW 2.8.1
     // Functionality: Conversion DB_ANY --> TO_Axis
     // Support: tech.team.motioncontrol@siemens.com
     // Note: Parameter comments are only available in language 'English (United States)'
     //--------------------------------------------------------------------------------
     // Change log table:
     // Version  Date        Expert in charge  Changes applied
     // 01.00.00 10.03.2020  RS                First released version
     //================================================================================
   END_REGION

   REGION EXECUTE
     IF #Execute AND NOT #statExecuteOld THEN
       // Copy parameter
       #instMC.Position := #Position;
       #instMC.Mode := #Mode;

       // Check axis type
       CASE TypeOfDB(#Axis) OF
         TO_POSITIONINGAXIS:
           #statAxisType := #POSITIONING_AXIS;
           #statAxis := #Axis;

         TO_SYNCHRONOUSAXIS:
           #statAxisType := #SYNCHRONOUS_AXIS;
           #statAxis := #Axis;

         TO_EXTERNALENCODER:
           #statAxisType := #EXTERNAL_ENCODER;
           #statAxis := #Axis;

         ELSE
           #statAxisType := #INVALID_AXIS;
           #statAxis := 0;
       END_CASE;

     ELSIF NOT #Execute AND (#statAxisType = #INVALID_AXIS) THEN
       #statAxisType := #IDLE;

       // Outputs
       #Done := FALSE;
       #Busy := FALSE;
       #CommandAborted := FALSE;
       #Error := FALSE;
       #ErrorID := 16#0000;
     END_IF;

     // Edge detection
     #statExecuteOld := #Execute;
   END_REGION

   CASE #statAxisType OF
     #IDLE:
       ;

     #POSITIONING_AXIS,
     #SYNCHRONOUS_AXIS,
     #EXTERNAL_ENCODER:
       REGION VALID_AXIS
         // Inputs
         #instMC.Execute := #Execute;

         // Call of MC instruction
         CASE #statAxisType OF
           #POSITIONING_AXIS:
             "LAnyAxis_UnpubHomePosAxis"(axis := #statAxis,
                                         instMC := #instMC);
           #SYNCHRONOUS_AXIS:
             "LAnyAxis_UnpubHomeSyncAxis"(axis := #statAxis,
                                          instMC := #instMC);
           #EXTERNAL_ENCODER:
             "LAnyAxis_UnpubHomeExtEncoder"(axis := #statAxis,
                                            instMC := #instMC);
         END_CASE;

         // Outputs
         #ReferenceMarkPosition := #instMC.ReferenceMarkPosition;
         #Done := #instMC.Done;
         #Busy := #instMC.Busy;
         #CommandAborted := #instMC.CommandAborted;
         #Error := #instMC.Error;
         #ErrorID := #instMC.ErrorId;

         // Status of MC instruction
         IF NOT #instMC.Done
           AND NOT #instMC.Busy
           AND NOT #instMC.CommandAborted
           AND NOT #instMC.Error
         THEN
           // Not active
           #statAxisType := #IDLE;
         END_IF;
       END_REGION

     ELSE
       REGION INVALID_AXIS
         // Outputs
         #Done := FALSE;
         #Busy := FALSE;
         #CommandAborted := FALSE;
         #Error := TRUE;
         #ErrorID := #ERROR_INVALID_TECHNOLOGY_OBJECT;
       END_REGION
   END_CASE;
END_FUNCTION_BLOCK

FUNCTION_BLOCK "LAnyAxis_MC_Halt"   // FB30003, SCL
TITLE = LAnyAxis_MC_Halt
{ S7_Optimized_Access := 'TRUE' }
AUTHOR : tech.team.motioncontrol@siemens.com
FAMILY : AnyAxis
VERSION : 1.0
// Support: tech.team.motioncontrol@siemens.com 
// See corresponding MC_ instruction in TIA Portal help (information system)
   VAR_INPUT
      Axis : DB_ANY;   // See corresponding parameter of MC_ instruction in TIA Portal help (information system)
      Execute : Bool;   // See corresponding parameter of MC_ instruction in TIA Portal help (information system)
      Deceleration : LReal := -1.0;   // See corresponding parameter of MC_ instruction in TIA Portal help (information system)
      Jerk : LReal := -1.0;   // See corresponding parameter of MC_ instruction in TIA Portal help (information system)
      AbortAcceleration : Bool;   // See corresponding parameter of MC_ instruction in TIA Portal help (information system)
   END_VAR
   VAR_OUTPUT
      Done : Bool;   // See corresponding parameter of MC_ instruction in TIA Portal help (information system)
      Busy : Bool;   // See corresponding parameter of MC_ instruction in TIA Portal help (information system)
      CommandAborted : Bool;   // See corresponding parameter of MC_ instruction in TIA Portal help (information system)
      Error : Bool;   // See corresponding parameter of MC_ instruction in TIA Portal help (information system)
      ErrorID : Word;   // See corresponding parameter of MC_ instruction in TIA Portal help (information system)
   END_VAR
   VAR
      instMC : MC_HALT;   // Instance of MC_Instruction
      statExecuteOld : Bool;   // Old value of execute
      statAxis : DB_ANY;   // Internal variable of axis
      statAxisType : Int;   // Actual state / axis type
   END_VAR
   VAR CONSTANT
      ERROR_INVALID_TECHNOLOGY_OBJECT : Word := 16#8002;   // See corresponding parameter of MC_ instruction in TIA Portal help (information system)
      IDLE : Int := 0;   // State idle
      INVALID_AXIS : Int := -1;   // Axis type: Invalid
      SPEED_AXIS : Int := 2;   // Axis type: Speed axis
      POSITIONING_AXIS : Int := 3;   // Axis type: Positioning axis
      SYNCHRONOUS_AXIS : Int := 4;   // Axis type: Synchronous axis
   END_VAR
BEGIN
   REGION HEADER
     //================================================================================
     // SIEMENS AG
     // (c)Copyright 2020 All Rights Reserved
     //--------------------------------------------------------------------------------
     // Library: LAnyAxis 
     // Tested with: S7-1515-2 PN
     // Engineering: TIA Portal V16
     // Restrictions: -
     // Requirements: S7-1500 FW 2.8.1
     // Functionality: Conversion DB_ANY --> TO_Axis
     // Support: tech.team.motioncontrol@siemens.com
     // Note: Parameter comments are only available in language 'English (United States)'
     //--------------------------------------------------------------------------------
     // Change log table:
     // Version  Date        Expert in charge  Changes applied
     // 01.00.00 10.03.2020  RS                First released version
     //================================================================================
   END_REGION

   REGION EXECUTE
     IF #Execute AND NOT #statExecuteOld THEN
       // Copy parameter
       #instMC.Deceleration := #Deceleration;
       #instMC.Jerk := #Jerk;
       #instMC.AbortAcceleration := #AbortAcceleration;

       // Check axis type
       CASE TypeOfDB(#Axis) OF
         TO_POSITIONINGAXIS:
           #statAxisType := #POSITIONING_AXIS;
           #statAxis := #Axis;

         TO_SYNCHRONOUSAXIS:
           #statAxisType := #SYNCHRONOUS_AXIS;
           #statAxis := #Axis;

         TO_SPEEDAXIS:
           #statAxisType := #SPEED_AXIS;
           #statAxis := #Axis;

         ELSE
           #statAxisType := #INVALID_AXIS;
           #statAxis := 0;
       END_CASE;

     ELSIF NOT #Execute AND (#statAxisType = #INVALID_AXIS) THEN
       #statAxisType := #IDLE;

       // Outputs
       #Done := FALSE;
       #Busy := FALSE;
       #CommandAborted := FALSE;
       #Error := FALSE;
       #ErrorID := 16#0000;
     END_IF;

     // Edge detection
     #statExecuteOld := #Execute;
   END_REGION

   CASE #statAxisType OF
     #IDLE:
       ;

     #POSITIONING_AXIS,
     #SYNCHRONOUS_AXIS,
     #SPEED_AXIS:
       REGION VALID_AXIS
         // Inputs
         #instMC.Execute := #Execute;

         // Call of MC instruction
         CASE #statAxisType OF
           #POSITIONING_AXIS:
             "LAnyAxis_UnpubHaltPosAxis"(axis := #statAxis,
                                         instMC := #instMC);
           #SYNCHRONOUS_AXIS:
             "LAnyAxis_UnpubHaltSyncAxis"(axis := #statAxis,
                                          instMC := #instMC);
           #SPEED_AXIS:
             #instMC(Axis := #statAxis);
         END_CASE;

         // Outputs
         #Done := #instMC.Done;
         #Busy := #instMC.Busy;
         #CommandAborted := #instMC.CommandAborted;
         #Error := #instMC.Error;
         #ErrorID := #instMC.ErrorId;

         // Status of MC instruction
         IF NOT #instMC.Done
           AND NOT #instMC.Busy
           AND NOT #instMC.CommandAborted
           AND NOT #instMC.Error
         THEN
           // Not active
           #statAxisType := #IDLE;
         END_IF;
       END_REGION

     ELSE
       REGION INVALID_AXIS
         // Outputs
         #Done := FALSE;
         #Busy := FALSE;
         #CommandAborted := FALSE;
         #Error := TRUE;
         #ErrorID := #ERROR_INVALID_TECHNOLOGY_OBJECT;
       END_REGION
   END_CASE;
END_FUNCTION_BLOCK

FUNCTION_BLOCK "LAnyAxis_MC_MoveAbsolute"   // FB30004, SCL
TITLE = LAnyAxis_MC_MoveAbsolute
{ S7_Optimized_Access := 'TRUE' }
AUTHOR : tech.team.motioncontrol@siemens.com
FAMILY : AnyAxis
VERSION : 1.0
// Support: tech.team.motioncontrol@siemens.com 
// See corresponding MC_ instruction in TIA Portal help (information system)
   VAR_INPUT
      Axis : DB_ANY;   // See corresponding parameter of MC_ instruction in TIA Portal help (information system)
      Execute : Bool;   // See corresponding parameter of MC_ instruction in TIA Portal help (information system)
      Position : LReal;   // See corresponding parameter of MC_ instruction in TIA Portal help (information system)
      Velocity : LReal := -1.0;   // See corresponding parameter of MC_ instruction in TIA Portal help (information system)
      Acceleration : LReal := -1.0;   // See corresponding parameter of MC_ instruction in TIA Portal help (information system)
      Deceleration : LReal := -1.0;   // See corresponding parameter of MC_ instruction in TIA Portal help (information system)
      Jerk : LReal := -1.0;   // See corresponding parameter of MC_ instruction in TIA Portal help (information system)
      Direction : Int := 1;   // See corresponding parameter of MC_ instruction in TIA Portal help (information system)
   END_VAR
   VAR_OUTPUT
      Done : Bool;   // See corresponding parameter of MC_ instruction in TIA Portal help (information system)
      Busy : Bool;   // See corresponding parameter of MC_ instruction in TIA Portal help (information system)
      CommandAborted : Bool;   // See corresponding parameter of MC_ instruction in TIA Portal help (information system)
      Error : Bool;   // See corresponding parameter of MC_ instruction in TIA Portal help (information system)
      ErrorID : Word;   // See corresponding parameter of MC_ instruction in TIA Portal help (information system)
   END_VAR
   VAR
      instMC : MC_MOVEABSOLUTE;   // Instance of MC_Instruction
      statExecuteOld : Bool;   // Old value of execute
      statAxis : DB_ANY;   // Internal variable of axis
      statAxisType : Int;   // Actual state / axis type
   END_VAR
   VAR CONSTANT
      ERROR_INVALID_TECHNOLOGY_OBJECT : Word := 16#8002;   // See corresponding parameter of MC_ instruction in TIA Portal help (information system)
      IDLE : Int := 0;   // State idle
      INVALID_AXIS : Int := -1;   // Axis type: Invalid
      EXTERNAL_ENCODER : Int := 1;   // Axis type: External encoder
      POSITIONING_AXIS : Int := 3;   // Axis type: Positioning axis
      SYNCHRONOUS_AXIS : Int := 4;   // Axis type: Synchronous axis
   END_VAR
BEGIN
   REGION HEADER
     //================================================================================
     // SIEMENS AG
     // (c)Copyright 2020 All Rights Reserved
     //--------------------------------------------------------------------------------
     // Library: LAnyAxis 
     // Tested with: S7-1515-2 PN
     // Engineering: TIA Portal V16
     // Restrictions: -
     // Requirements: S7-1500 FW 2.8.1
     // Functionality: Conversion DB_ANY --> TO_Axis
     // Support: tech.team.motioncontrol@siemens.com
     // Note: Parameter comments are only available in language 'English (United States)'
     //--------------------------------------------------------------------------------
     // Change log table:
     // Version  Date        Expert in charge  Changes applied
     // 01.00.00 10.03.2020  RS                First released version
     //================================================================================
   END_REGION

   REGION EXECUTE
     IF #Execute AND NOT #statExecuteOld THEN
       // Copy parameter
       #instMC.Position := #Position;
       #instMC.Velocity := #Velocity;
       #instMC.Acceleration := #Acceleration;
       #instMC.Deceleration := #Deceleration;
       #instMC.Jerk := #Jerk;
       #instMC.Direction := #Direction;

       // Check axis type
       CASE TypeOfDB(#Axis) OF
         TO_POSITIONINGAXIS:
           #statAxisType := #POSITIONING_AXIS;
           #statAxis := #Axis;

         TO_SYNCHRONOUSAXIS:
           #statAxisType := #SYNCHRONOUS_AXIS;
           #statAxis := #Axis;

         ELSE
           #statAxisType := #INVALID_AXIS;
           #statAxis := 0;
       END_CASE;

     ELSIF NOT #Execute AND (#statAxisType = #INVALID_AXIS) THEN
       #statAxisType := #IDLE;

       // Outputs
       #Done := FALSE;
       #Busy := FALSE;
       #CommandAborted := FALSE;
       #Error := FALSE;
       #ErrorID := 16#0000;
     END_IF;

     // Edge detection
     #statExecuteOld := #Execute;
   END_REGION

   CASE #statAxisType OF
     #IDLE:
       ;

     #POSITIONING_AXIS,
     #SYNCHRONOUS_AXIS:
       REGION VALID_AXIS
         // Inputs
         #instMC.Execute := #Execute;

         // Call of MC instruction
         CASE #statAxisType OF
           #POSITIONING_AXIS:
             #instMC(Axis := #statAxis);
           #SYNCHRONOUS_AXIS:
             "LAnyAxis_UnpubMoveAbsoluteSyncAxis"(axis := #statAxis,
                                                  instMC := #instMC);
         END_CASE;

         // Outputs
         #Done := #instMC.Done;
         #Busy := #instMC.Busy;
         #CommandAborted := #instMC.CommandAborted;
         #Error := #instMC.Error;
         #ErrorID := #instMC.ErrorId;

         // Status of MC instruction
         IF NOT #instMC.Done
           AND NOT #instMC.Busy
           AND NOT #instMC.CommandAborted
           AND NOT #instMC.Error
         THEN
           // Not active
           #statAxisType := #IDLE;
         END_IF;
       END_REGION

     ELSE
       REGION INVALID_AXIS
         // Outputs
         #Done := FALSE;
         #Busy := FALSE;
         #CommandAborted := FALSE;
         #Error := TRUE;
         #ErrorID := #ERROR_INVALID_TECHNOLOGY_OBJECT;
       END_REGION
   END_CASE;
END_FUNCTION_BLOCK

FUNCTION_BLOCK "LAnyAxis_MC_MoveRelative"   // FB30005, SCL
TITLE = LAnyAxis_MC_MoveRelative
{ S7_Optimized_Access := 'TRUE' }
AUTHOR : tech.team.motioncontrol@siemens.com
FAMILY : AnyAxis
VERSION : 1.0
// Support: tech.team.motioncontrol@siemens.com 
// See corresponding MC_ instruction in TIA Portal help (information system)
   VAR_INPUT
      Axis : DB_ANY;   // See corresponding parameter of MC_ instruction in TIA Portal help (information system)
      Execute : Bool;   // See corresponding parameter of MC_ instruction in TIA Portal help (information system)
      Distance : LReal;   // See corresponding parameter of MC_ instruction in TIA Portal help (information system)
      Velocity : LReal := -1.0;   // See corresponding parameter of MC_ instruction in TIA Portal help (information system)
      Acceleration : LReal := -1.0;   // See corresponding parameter of MC_ instruction in TIA Portal help (information system)
      Deceleration : LReal := -1.0;   // See corresponding parameter of MC_ instruction in TIA Portal help (information system)
      Jerk : LReal := -1.0;   // See corresponding parameter of MC_ instruction in TIA Portal help (information system)
   END_VAR
   VAR_OUTPUT
      Done : Bool;   // See corresponding parameter of MC_ instruction in TIA Portal help (information system)
      Busy : Bool;   // See corresponding parameter of MC_ instruction in TIA Portal help (information system)
      CommandAborted : Bool;   // See corresponding parameter of MC_ instruction in TIA Portal help (information system)
      Error : Bool;   // See corresponding parameter of MC_ instruction in TIA Portal help (information system)
      ErrorID : Word;   // See corresponding parameter of MC_ instruction in TIA Portal help (information system)
   END_VAR
   VAR
      instMC : MC_MOVERELATIVE;   // Instance of MC_Instruction
      statExecuteOld : Bool;   // Old value of execute
      statAxis : DB_ANY;   // Internal variable of axis
      statAxisType : Int;   // Actual state / axis type
   END_VAR
   VAR CONSTANT
      ERROR_INVALID_TECHNOLOGY_OBJECT : Word := 16#8002;   // See corresponding parameter of MC_ instruction in TIA Portal help (information system)
      IDLE : Int := 0;   // State idle
      INVALID_AXIS : Int := -1;   // Axis type: Invalid
      POSITIONING_AXIS : Int := 3;   // Axis type: Positioning axis
      SYNCHRONOUS_AXIS : Int := 4;   // Axis type: Synchronous axis
   END_VAR
BEGIN
   REGION HEADER
     //================================================================================
     // SIEMENS AG
     // (c)Copyright 2020 All Rights Reserved
     //--------------------------------------------------------------------------------
     // Library: LAnyAxis 
     // Tested with: S7-1515-2 PN
     // Engineering: TIA Portal V16
     // Restrictions: -
     // Requirements: S7-1500 FW 2.8.1
     // Functionality: Conversion DB_ANY --> TO_Axis
     // Support: tech.team.motioncontrol@siemens.com
     // Note: Parameter comments are only available in language 'English (United States)'
     //--------------------------------------------------------------------------------
     // Change log table:
     // Version  Date        Expert in charge  Changes applied
     // 01.00.00 10.03.2020  RS                First released version
     //================================================================================
   END_REGION

   REGION EXECUTE
     IF #Execute AND NOT #statExecuteOld THEN
       // Copy parameter
       #instMC.Distance := #Distance;
       #instMC.Velocity := #Velocity;
       #instMC.Acceleration := #Acceleration;
       #instMC.Deceleration := #Deceleration;
       #instMC.Jerk := #Jerk;

       // Check axis type
       CASE TypeOfDB(#Axis) OF
         TO_POSITIONINGAXIS:
           #statAxisType := #POSITIONING_AXIS;
           #statAxis := #Axis;

         TO_SYNCHRONOUSAXIS:
           #statAxisType := #SYNCHRONOUS_AXIS;
           #statAxis := #Axis;

         ELSE
           #statAxisType := #INVALID_AXIS;
           #statAxis := 0;
       END_CASE;

     ELSIF NOT #Execute AND (#statAxisType = #INVALID_AXIS) THEN
       #statAxisType := #IDLE;

       // Outputs
       #Done := FALSE;
       #Busy := FALSE;
       #CommandAborted := FALSE;
       #Error := FALSE;
       #ErrorID := 16#0000;
     END_IF;

     // Edge detection
     #statExecuteOld := #Execute;
   END_REGION

   CASE #statAxisType OF
     #IDLE:
       ;

     #POSITIONING_AXIS,
     #SYNCHRONOUS_AXIS:
       REGION VALID_AXIS
         // Inputs
         #instMC.Execute := #Execute;

         // Call of MC instruction
         CASE #statAxisType OF
           #POSITIONING_AXIS:
             #instMC(Axis := #statAxis);
           #SYNCHRONOUS_AXIS:
             "LAnyAxis_UnpubMoveRelativeSyncAxis"(axis := #statAxis,
                                                  instMC := #instMC);
         END_CASE;

         // Outputs
         #Done := #instMC.Done;
         #Busy := #instMC.Busy;
         #CommandAborted := #instMC.CommandAborted;
         #Error := #instMC.Error;
         #ErrorID := #instMC.ErrorId;

         // Status of MC instruction
         IF NOT #instMC.Done
           AND NOT #instMC.Busy
           AND NOT #instMC.CommandAborted
           AND NOT #instMC.Error
         THEN
           // Not active
           #statAxisType := #IDLE;
         END_IF;
       END_REGION

     ELSE
       REGION INVALID_AXIS
         // Outputs
         #Done := FALSE;
         #Busy := FALSE;
         #CommandAborted := FALSE;
         #Error := TRUE;
         #ErrorID := #ERROR_INVALID_TECHNOLOGY_OBJECT;
       END_REGION
   END_CASE;
END_FUNCTION_BLOCK

FUNCTION_BLOCK "LAnyAxis_MC_MoveVelocity"   // FB30006, SCL
TITLE = LAnyAxis_MC_MoveVelocity
{ S7_Optimized_Access := 'TRUE' }
AUTHOR : tech.team.motioncontrol@siemens.com
FAMILY : AnyAxis
VERSION : 1.0
// Support: tech.team.motioncontrol@siemens.com 
// See corresponding MC_ instruction in TIA Portal help (information system)
   VAR_INPUT
      Axis : DB_ANY;   // See corresponding parameter of MC_ instruction in TIA Portal help (information system)
      Execute : Bool;   // See corresponding parameter of MC_ instruction in TIA Portal help (information system)
      Velocity : LReal := 100.0;   // See corresponding parameter of MC_ instruction in TIA Portal help (information system)
      Acceleration : LReal := -1.0;   // See corresponding parameter of MC_ instruction in TIA Portal help (information system)
      Deceleration : LReal := -1.0;   // See corresponding parameter of MC_ instruction in TIA Portal help (information system)
      Jerk : LReal := -1.0;   // See corresponding parameter of MC_ instruction in TIA Portal help (information system)
      Direction : Int;   // See corresponding parameter of MC_ instruction in TIA Portal help (information system)
      Current : Bool;   // See corresponding parameter of MC_ instruction in TIA Portal help (information system)
      PositionControlled : Bool := TRUE;   // See corresponding parameter of MC_ instruction in TIA Portal help (information system)
   END_VAR
   VAR_OUTPUT
      InVelocity : Bool;   // See corresponding parameter of MC_ instruction in TIA Portal help (information system)
      Busy : Bool;   // See corresponding parameter of MC_ instruction in TIA Portal help (information system)
      CommandAborted : Bool;   // See corresponding parameter of MC_ instruction in TIA Portal help (information system)
      Error : Bool;   // See corresponding parameter of MC_ instruction in TIA Portal help (information system)
      ErrorID : Word;   // See corresponding parameter of MC_ instruction in TIA Portal help (information system)
   END_VAR
   VAR
      instMC : MC_MOVEVELOCITY;   // Instance of MC_Instruction
      statExecuteOld : Bool;   // Old value of execute
      statAxis : DB_ANY;   // Internal variable of axis
      statAxisType : Int;   // Actual state / axis type
   END_VAR
   VAR CONSTANT
      ERROR_INVALID_TECHNOLOGY_OBJECT : Word := 16#8002;   // See corresponding parameter of MC_ instruction in TIA Portal help (information system)
      IDLE : Int := 0;   // State idle
      INVALID_AXIS : Int := -1;   // Axis type: Invalid
      SPEED_AXIS : Int := 2;   // Axis type: Speed axis
      POSITIONING_AXIS : Int := 3;   // Axis type: Positioning axis
      SYNCHRONOUS_AXIS : Int := 4;   // Axis type: Synchronous axis
   END_VAR
BEGIN
   REGION HEADER
     //================================================================================
     // SIEMENS AG
     // (c)Copyright 2020 All Rights Reserved
     //--------------------------------------------------------------------------------
     // Library: LAnyAxis 
     // Tested with: S7-1515-2 PN
     // Engineering: TIA Portal V16
     // Restrictions: -
     // Requirements: S7-1500 FW 2.8.1
     // Functionality: Conversion DB_ANY --> TO_Axis
     // Support: tech.team.motioncontrol@siemens.com
     // Note: Parameter comments are only available in language 'English (United States)'
     //--------------------------------------------------------------------------------
     // Change log table:
     // Version  Date        Expert in charge  Changes applied
     // 01.00.00 10.03.2020  RS                First released version
     //================================================================================
   END_REGION

   REGION EXECUTE
     IF #Execute AND NOT #statExecuteOld THEN
       // Copy parameter
       #instMC.Velocity := #Velocity;
       #instMC.Acceleration := #Acceleration;
       #instMC.Deceleration := #Deceleration;
       #instMC.Jerk := #Jerk;
       #instMC.Direction := #Direction;
       #instMC.Current := #Current;
       #instMC.PositionControlled := #PositionControlled;

       // Check axis type
       CASE TypeOfDB(#Axis) OF
         TO_POSITIONINGAXIS:
           #statAxisType := #POSITIONING_AXIS;
           #statAxis := #Axis;

         TO_SYNCHRONOUSAXIS:
           #statAxisType := #SYNCHRONOUS_AXIS;
           #statAxis := #Axis;

         TO_SPEEDAXIS:
           #statAxisType := #SPEED_AXIS;
           #statAxis := #Axis;

         ELSE
           #statAxisType := #INVALID_AXIS;
           #statAxis := 0;
       END_CASE;

     ELSIF NOT #Execute AND (#statAxisType = #INVALID_AXIS) THEN
       #statAxisType := #IDLE;

       // Outputs
       #InVelocity := FALSE;
       #Busy := FALSE;
       #CommandAborted := FALSE;
       #Error := FALSE;
       #ErrorID := 16#0000;
     END_IF;

     // Edge detection
     #statExecuteOld := #Execute;
   END_REGION

   CASE #statAxisType OF
     #IDLE:
       ;

     #POSITIONING_AXIS,
     #SYNCHRONOUS_AXIS,
     #SPEED_AXIS:
       REGION VALID_AXIS
         // Inputs
         #instMC.Execute := #Execute;

         // Call of MC instruction
         CASE #statAxisType OF
           #POSITIONING_AXIS:
             "LAnyAxis_UnpubMoveVelocityPosAxis"(axis := #statAxis,
                                                 instMC := #instMC);
           #SYNCHRONOUS_AXIS:
             "LAnyAxis_UnpubMoveVelocitySyncAxis"(axis := #statAxis,
                                                  instMC := #instMC);
           #SPEED_AXIS:
             #instMC(Axis := #statAxis);
         END_CASE;

         // Outputs
         #InVelocity := #instMC.InVelocity;
         #Busy := #instMC.Busy;
         #CommandAborted := #instMC.CommandAborted;
         #Error := #instMC.Error;
         #ErrorID := #instMC.ErrorId;

         // Status of MC instruction
         IF NOT #instMC.Busy
           AND NOT #instMC.CommandAborted
           AND NOT #instMC.Error
         THEN
           // Not active
           #statAxisType := #IDLE;
         END_IF;
       END_REGION

     ELSE
       REGION INVALID_AXIS
         // Outputs
         #InVelocity := FALSE;
         #Busy := FALSE;
         #CommandAborted := FALSE;
         #Error := TRUE;
         #ErrorID := #ERROR_INVALID_TECHNOLOGY_OBJECT;
       END_REGION
   END_CASE;
END_FUNCTION_BLOCK

FUNCTION_BLOCK "LAnyAxis_MC_MoveJog"   // FB30007, SCL
TITLE = LAnyAxis_MC_MoveJog
{ S7_Optimized_Access := 'TRUE' }
AUTHOR : tech.team.motioncontrol@siemens.com
FAMILY : AnyAxis
VERSION : 1.0
// Support: tech.team.motioncontrol@siemens.com 
// See corresponding MC_ instruction in TIA Portal help (information system)
   VAR_INPUT
      Axis : DB_ANY;   // See corresponding parameter of MC_ instruction in TIA Portal help (information system)
      JogForward : Bool;   // See corresponding parameter of MC_ instruction in TIA Portal help (information system)
      JogBackward : Bool;   // See corresponding parameter of MC_ instruction in TIA Portal help (information system)
      Velocity : LReal := 100.0;   // See corresponding parameter of MC_ instruction in TIA Portal help (information system)
      Acceleration : LReal := -1.0;   // See corresponding parameter of MC_ instruction in TIA Portal help (information system)
      Deceleration : LReal := -1.0;   // See corresponding parameter of MC_ instruction in TIA Portal help (information system)
      Jerk : LReal := -1.0;   // See corresponding parameter of MC_ instruction in TIA Portal help (information system)
      PositionControlled : Bool := TRUE;   // See corresponding parameter of MC_ instruction in TIA Portal help (information system)
   END_VAR
   VAR_OUTPUT
      InVelocity : Bool;   // See corresponding parameter of MC_ instruction in TIA Portal help (information system)
      Busy : Bool;   // See corresponding parameter of MC_ instruction in TIA Portal help (information system)
      CommandAborted : Bool;   // See corresponding parameter of MC_ instruction in TIA Portal help (information system)
      Error : Bool;   // See corresponding parameter of MC_ instruction in TIA Portal help (information system)
      ErrorID : Word;   // See corresponding parameter of MC_ instruction in TIA Portal help (information system)
   END_VAR
   VAR
      instMC : MC_MOVEJOG;   // Instance of MC_Instruction
      statAxis : DB_ANY;   // Internal variable of axis
      statAxisType : Int;   // Actual state / axis type
   END_VAR
   VAR CONSTANT
      ERROR_INVALID_TECHNOLOGY_OBJECT : Word := 16#8002;   // See corresponding parameter of MC_ instruction in TIA Portal help (information system)
      IDLE : Int := 0;   // State idle
      INVALID_AXIS : Int := -1;   // Axis type: Invalid
      SPEED_AXIS : Int := 2;   // Axis type: Speed axis
      POSITIONING_AXIS : Int := 3;   // Axis type: Positioning axis
      SYNCHRONOUS_AXIS : Int := 4;   // Axis type: Synchronous axis
   END_VAR
BEGIN
   REGION HEADER
     //================================================================================
     // SIEMENS AG
     // (c)Copyright 2020 All Rights Reserved
     //--------------------------------------------------------------------------------
     // Library: LAnyAxis 
     // Tested with: S7-1515-2 PN
     // Engineering: TIA Portal V16
     // Restrictions: -
     // Requirements: S7-1500 FW 2.8.1
     // Functionality: Conversion DB_ANY --> TO_Axis
     // Support: tech.team.motioncontrol@siemens.com
     // Note: Parameter comments are only available in language 'English (United States)'
     //--------------------------------------------------------------------------------
     // Change log table:
     // Version  Date        Expert in charge  Changes applied
     // 01.00.00 10.03.2020  RS                First released version
     //================================================================================
   END_REGION

   REGION ENABLE
     IF (#statAxisType = #IDLE) AND (#JogForward OR #JogBackward) THEN
       // Check axis type
       CASE TypeOfDB(#Axis) OF
         TO_POSITIONINGAXIS:
           #statAxisType := #POSITIONING_AXIS;
           #statAxis := #Axis;

         TO_SYNCHRONOUSAXIS:
           #statAxisType := #SYNCHRONOUS_AXIS;
           #statAxis := #Axis;

         TO_SPEEDAXIS:
           #statAxisType := #SPEED_AXIS;
           #statAxis := #Axis;

         ELSE
           #statAxisType := #INVALID_AXIS;
           #statAxis := 0;
       END_CASE;

     ELSIF NOT #JogForward AND NOT #JogBackward AND (#statAxisType = #INVALID_AXIS) THEN
       #statAxisType := #IDLE;

       // Outputs
       #InVelocity := FALSE;
       #Busy := FALSE;
       #CommandAborted := FALSE;
       #Error := FALSE;
       #ErrorID := 16#0000;
     END_IF;
   END_REGION

   CASE #statAxisType OF
     #IDLE:
       ;

     #POSITIONING_AXIS,
     #SYNCHRONOUS_AXIS,
     #SPEED_AXIS:
       REGION VALID_AXIS
         // Inputs
         #instMC.JogForward := #JogForward;
         #instMC.JogBackward := #JogBackward;
         #instMC.Velocity := #Velocity;
         #instMC.Acceleration := #Acceleration;
         #instMC.Deceleration := #Deceleration;
         #instMC.Jerk := #Jerk;
         #instMC.PositionControlled := #PositionControlled;

         // Call of MC instruction
         CASE #statAxisType OF
           #POSITIONING_AXIS:
             "LAnyAxis_UnpubMoveJogPosAxis"(axis := #statAxis,
                                            instMC := #instMC);
           #SYNCHRONOUS_AXIS:
             "LAnyAxis_UnpubMoveJogSyncAxis"(axis := #statAxis,
                                             instMC := #instMC);
           #SPEED_AXIS:
             #instMC(Axis := #statAxis);
         END_CASE;

         // Outputs
         #InVelocity := #instMC.InVelocity;
         #Busy := #instMC.Busy;
         #CommandAborted := #instMC.CommandAborted;
         #Error := #instMC.Error;
         #ErrorID := #instMC.ErrorId;

         // Status of MC instruction
         IF NOT #instMC.Busy
           AND NOT #instMC.Error
           AND NOT #instMC.CommandAborted
         THEN
           // Not active
           #statAxisType := #IDLE;
         END_IF;
       END_REGION

     ELSE
       REGION INVALID_AXIS
         // Outputs
         #InVelocity := FALSE;
         #Busy := FALSE;
         #CommandAborted := FALSE;
         #Error := TRUE;
         #ErrorID := #ERROR_INVALID_TECHNOLOGY_OBJECT;
       END_REGION
   END_CASE;
END_FUNCTION_BLOCK

FUNCTION_BLOCK "LAnyAxis_MC_MoveSuperimposed"   // FB30008, SCL
TITLE = LAnyAxis_MC_MoveSuperimposed
{ S7_Optimized_Access := 'TRUE' }
AUTHOR : tech.team.motioncontrol@siemens.com
FAMILY : AnyAxis
VERSION : 1.0
// Support: tech.team.motioncontrol@siemens.com 
// See corresponding MC_ instruction in TIA Portal help (information system)
   VAR_INPUT
      Axis : DB_ANY;   // See corresponding parameter of MC_ instruction in TIA Portal help (information system)
      Execute : Bool;   // See corresponding parameter of MC_ instruction in TIA Portal help (information system)
      Distance : LReal;   // See corresponding parameter of MC_ instruction in TIA Portal help (information system)
      VelocityDiff : LReal := -1.0;   // See corresponding parameter of MC_ instruction in TIA Portal help (information system)
      Acceleration : LReal := -1.0;   // See corresponding parameter of MC_ instruction in TIA Portal help (information system)
      Deceleration : LReal := -1.0;   // See corresponding parameter of MC_ instruction in TIA Portal help (information system)
      Jerk : LReal := -1.0;   // See corresponding parameter of MC_ instruction in TIA Portal help (information system)
   END_VAR
   VAR_OUTPUT
      Done : Bool;   // See corresponding parameter of MC_ instruction in TIA Portal help (information system)
      Busy : Bool;   // See corresponding parameter of MC_ instruction in TIA Portal help (information system)
      CommandAborted : Bool;   // See corresponding parameter of MC_ instruction in TIA Portal help (information system)
      Error : Bool;   // See corresponding parameter of MC_ instruction in TIA Portal help (information system)
      ErrorID : Word;   // See corresponding parameter of MC_ instruction in TIA Portal help (information system)
   END_VAR
   VAR
      instMC : MC_MOVESUPERIMPOSED;   // Instance of MC_Instruction
      statExecuteOld : Bool;   // Old value of execute
      statAxis : DB_ANY;   // Internal variable of axis
      statAxisType : Int;   // Actual state / axis type
   END_VAR
   VAR CONSTANT
      ERROR_INVALID_TECHNOLOGY_OBJECT : Word := 16#8002;   // See corresponding parameter of MC_ instruction in TIA Portal help (information system)
      IDLE : Int := 0;   // State idle
      INVALID_AXIS : Int := -1;   // Axis type: Invalid
      POSITIONING_AXIS : Int := 3;   // Axis type: Positioning axis
      SYNCHRONOUS_AXIS : Int := 4;   // Axis type: Synchronous axis
   END_VAR
BEGIN
   REGION HEADER
     //================================================================================
     // SIEMENS AG
     // (c)Copyright 2020 All Rights Reserved
     //--------------------------------------------------------------------------------
     // Library: LAnyAxis 
     // Tested with: S7-1515-2 PN
     // Engineering: TIA Portal V16
     // Restrictions: -
     // Requirements: S7-1500 FW 2.8.1
     // Functionality: Conversion DB_ANY --> TO_Axis
     // Support: tech.team.motioncontrol@siemens.com
     // Note: Parameter comments are only available in language 'English (United States)'
     //--------------------------------------------------------------------------------
     // Change log table:
     // Version  Date        Expert in charge  Changes applied
     // 01.00.00 10.03.2020  RS                First released version
     //================================================================================
   END_REGION

   REGION EXECUTE
     IF #Execute AND NOT #statExecuteOld THEN
       // Copy parameter
       #instMC.Distance := #Distance;
       #instMC.VelocityDiff := #VelocityDiff;
       #instMC.Acceleration := #Acceleration;
       #instMC.Deceleration := #Deceleration;
       #instMC.Jerk := #Jerk;

       // Check axis type
       CASE TypeOfDB(#Axis) OF
         TO_POSITIONINGAXIS:
           #statAxisType := #POSITIONING_AXIS;
           #statAxis := #Axis;

         TO_SYNCHRONOUSAXIS:
           #statAxisType := #SYNCHRONOUS_AXIS;
           #statAxis := #Axis;

         ELSE
           #statAxisType := #INVALID_AXIS;
           #statAxis := 0;
       END_CASE;

     ELSIF NOT #Execute AND (#statAxisType = #INVALID_AXIS) THEN
       #statAxisType := #IDLE;

       // Outputs
       #Done := FALSE;
       #Busy := FALSE;
       #CommandAborted := FALSE;
       #Error := FALSE;
       #ErrorID := 16#0000;
     END_IF;

     // Edge detection
     #statExecuteOld := #Execute;
   END_REGION

   CASE #statAxisType OF
     #IDLE:
       ;

     #POSITIONING_AXIS,
     #SYNCHRONOUS_AXIS:
       REGION VALID_AXIS
         // Inputs
         #instMC.Execute := #Execute;

         // Call of MC instruction
         CASE #statAxisType OF
           #POSITIONING_AXIS:
             #instMC(Axis := #statAxis);
           #SYNCHRONOUS_AXIS:
             "LAnyAxis_UnpubMoveSuperimposedSyncAxis"(axis := #statAxis,
                                                      instMC := #instMC);
         END_CASE;

         // Outputs
         #Done := #instMC.Done;
         #Busy := #instMC.Busy;
         #CommandAborted := #instMC.CommandAborted;
         #Error := #instMC.Error;
         #ErrorID := #instMC.ErrorId;

         // Status of MC instruction
         IF NOT #instMC.Done
           AND NOT #instMC.Busy
           AND NOT #instMC.CommandAborted
           AND NOT #instMC.Error
         THEN
           // Not active
           #statAxisType := #IDLE;
         END_IF;
       END_REGION

     ELSE
       REGION INVALID_AXIS
         // Outputs
         #Done := FALSE;
         #Busy := FALSE;
         #CommandAborted := FALSE;
         #Error := TRUE;
         #ErrorID := #ERROR_INVALID_TECHNOLOGY_OBJECT;
       END_REGION
   END_CASE;
END_FUNCTION_BLOCK

FUNCTION_BLOCK "LAnyAxis_MC_SetAxisSTW"   // FB30011, SCL
TITLE = LAnyAxis_MC_SetAxisSTW
{ S7_Optimized_Access := 'TRUE' }
AUTHOR : tech.team.motioncontrol@siemens.com
FAMILY : AnyAxis
VERSION : 1.0
// Support: tech.team.motioncontrol@siemens.com 
// See corresponding MC_ instruction in TIA Portal help (information system)
   VAR_INPUT
      Axis : DB_ANY;   // See corresponding parameter of MC_ instruction in TIA Portal help (information system)
      Execute : Bool;   // See corresponding parameter of MC_ instruction in TIA Portal help (information system)
      STW1 : Word;   // See corresponding parameter of MC_ instruction in TIA Portal help (information system)
      STW1BitMask : Word;   // See corresponding parameter of MC_ instruction in TIA Portal help (information system)
      STW2 : Word;   // See corresponding parameter of MC_ instruction in TIA Portal help (information system)
      STW2BitMask : Word;   // See corresponding parameter of MC_ instruction in TIA Portal help (information system)
   END_VAR
   VAR_OUTPUT
      Done : Bool;   // See corresponding parameter of MC_ instruction in TIA Portal help (information system)
      Busy : Bool;   // See corresponding parameter of MC_ instruction in TIA Portal help (information system)
      CommandAborted : Bool;   // See corresponding parameter of MC_ instruction in TIA Portal help (information system)
      Error : Bool;   // See corresponding parameter of MC_ instruction in TIA Portal help (information system)
      ErrorID : Word;   // See corresponding parameter of MC_ instruction in TIA Portal help (information system)
   END_VAR
   VAR
      instMC : MC_SETAXISSTW;   // Instance of MC_Instruction
      statExecuteOld : Bool;   // Old value of execute
      statAxis : DB_ANY;   // Internal variable of axis
      statAxisType : Int;   // Actual state / axis type
   END_VAR
   VAR CONSTANT
      ERROR_INVALID_TECHNOLOGY_OBJECT : Word := 16#8002;   // See corresponding parameter of MC_ instruction in TIA Portal help (information system)
      IDLE : Int := 0;   // State idle
      INVALID_AXIS : Int := -1;   // Axis type: Invalid
      SPEED_AXIS : Int := 2;   // Axis type: Speed axis
      POSITIONING_AXIS : Int := 3;   // Axis type: Positioning axis
      SYNCHRONOUS_AXIS : Int := 4;   // Axis type: Synchronous axis
   END_VAR
BEGIN
   REGION HEADER
     //================================================================================
     // SIEMENS AG
     // (c)Copyright 2020 All Rights Reserved
     //--------------------------------------------------------------------------------
     // Library: LAnyAxis 
     // Tested with: S7-1515-2 PN
     // Engineering: TIA Portal V16
     // Restrictions: -
     // Requirements: S7-1500 FW 2.8.1
     // Functionality: Conversion DB_ANY --> TO_Axis
     // Support: tech.team.motioncontrol@siemens.com
     // Note: Parameter comments are only available in language 'English (United States)'
     //--------------------------------------------------------------------------------
     // Change log table:
     // Version  Date        Expert in charge  Changes applied
     // 01.00.00 10.03.2020  RS                First released version
     //================================================================================
   END_REGION

   REGION EXECUTE
     IF #Execute AND NOT #statExecuteOld THEN
       // Copy parameter
       #instMC.STW1 := #STW1;
       #instMC.STW1BitMask := #STW1BitMask;
       #instMC.STW2 := #STW2;
       #instMC.STW2BitMask := #STW2BitMask;

       // Check axis type
       CASE TypeOfDB(#Axis) OF
         TO_POSITIONINGAXIS:
           #statAxisType := #POSITIONING_AXIS;
           #statAxis := #Axis;

         TO_SYNCHRONOUSAXIS:
           #statAxisType := #SYNCHRONOUS_AXIS;
           #statAxis := #Axis;

         TO_SPEEDAXIS:
           #statAxisType := #SPEED_AXIS;
           #statAxis := #Axis;

         ELSE
           #statAxisType := #INVALID_AXIS;
           #statAxis := 0;
       END_CASE;

     ELSIF NOT #Execute AND (#statAxisType = #INVALID_AXIS) THEN
       #statAxisType := #IDLE;

       // Outputs
       #Done := FALSE;
       #Busy := FALSE;
       #CommandAborted := FALSE;
       #Error := FALSE;
       #ErrorID := 16#0000;
     END_IF;

     // Edge detection
     #statExecuteOld := #Execute;
   END_REGION

   CASE #statAxisType OF
     #IDLE:
       ;

     #POSITIONING_AXIS,
     #SYNCHRONOUS_AXIS,
     #SPEED_AXIS:
       REGION VALID_AXIS
         // Inputs
         #instMC.Execute := #Execute;

         // Call of MC instruction
         CASE #statAxisType OF
           #POSITIONING_AXIS:
             "LAnyAxis_UnpubSetAxisSTWPosAxis"(axis := #statAxis,
                                               instMC := #instMC);
           #SYNCHRONOUS_AXIS:
             "LAnyAxis_UnpubSetAxisSTWSyncAxis"(axis := #statAxis,
                                                instMC := #instMC);
           #SPEED_AXIS:
             #instMC(Axis := #statAxis);
         END_CASE;

         // Outputs
         #Done := #instMC.Done;
         #Busy := #instMC.Busy;
         #CommandAborted := #instMC.CommandAborted;
         #Error := #instMC.Error;
         #ErrorID := #instMC.ErrorId;

         // Status of MC instruction
         IF NOT #instMC.Done
           AND NOT #instMC.Busy
           AND NOT #instMC.CommandAborted
           AND NOT #instMC.Error
         THEN
           // Not active
           #statAxisType := #IDLE;
         END_IF;
       END_REGION

     ELSE
       REGION INVALID_AXIS
         // Outputs
         #Done := FALSE;
         #Busy := FALSE;
         #CommandAborted := FALSE;
         #Error := TRUE;
         #ErrorID := #ERROR_INVALID_TECHNOLOGY_OBJECT;
       END_REGION
   END_CASE;
END_FUNCTION_BLOCK

// folder: LAnyAxis_Blocks/InternalSubBlocks/MC_Halt

FUNCTION "LAnyAxis_UnpubHaltPosAxis" : Void   // FC30003, SCL
TITLE = LAnyAxis_UnpubHaltPosAxis
{ S7_Optimized_Access := 'TRUE' }
AUTHOR : tech.team.motioncontrol@siemens.com
FAMILY : AnyAxis
VERSION : 1.0
// Support: tech.team.motioncontrol@siemens.com
   VAR_INPUT
      axis : TO_PositioningAxis;   // Axis specification
   END_VAR
   VAR_IN_OUT
      instMC : MC_HALT;   // Instance of MC_Instruction
   END_VAR
   // Ret_Val : No return value
BEGIN
   // Call of MC_Instruction
   #instMC(Axis := #axis);
END_FUNCTION

FUNCTION "LAnyAxis_UnpubHaltSyncAxis" : Void   // FC30005, SCL
TITLE = LAnyAxis_UnpubHaltSyncAxis
{ S7_Optimized_Access := 'TRUE' }
AUTHOR : tech.team.motioncontrol@siemens.com
FAMILY : AnyAxis
VERSION : 1.0
// Support: tech.team.motioncontrol@siemens.com
   VAR_INPUT
      axis : TO_SynchronousAxis;   // Axis specification
   END_VAR
   VAR_IN_OUT
      instMC : MC_HALT;   // Instance of MC_Instruction
   END_VAR
   // Ret_Val : No return value
BEGIN
   // Call of MC_Instruction
   #instMC(Axis := #axis);
END_FUNCTION

// folder: LAnyAxis_Blocks/InternalSubBlocks/MC_Home

FUNCTION "LAnyAxis_UnpubHomeExtEncoder" : Void   // FC30058, SCL
TITLE = LAnyAxis_UnpubHomeExtEncoder
{ S7_Optimized_Access := 'TRUE' }
AUTHOR : tech.team.motioncontrol@siemens.com
FAMILY : AnyAxis
VERSION : 1.0
// Support: tech.team.motioncontrol@siemens.com
   VAR_INPUT
      axis : TO_ExternalEncoder;   // Axis specification
   END_VAR
   VAR_IN_OUT
      instMC : MC_HOME;   // Instance of MC_Instruction
   END_VAR
   // Ret_Val : No return value
BEGIN
   // Call of MC_Instruction
   #instMC(Axis := #axis);
END_FUNCTION

FUNCTION "LAnyAxis_UnpubHomePosAxis" : Void   // FC30059, SCL
TITLE = LAnyAxis_UnpubHomePosAxis
{ S7_Optimized_Access := 'TRUE' }
AUTHOR : tech.team.motioncontrol@siemens.com
FAMILY : AnyAxis
VERSION : 1.0
// Support: tech.team.motioncontrol@siemens.com
   VAR_INPUT
      axis : TO_PositioningAxis;   // Axis specification
   END_VAR
   VAR_IN_OUT
      instMC : MC_HOME;   // Instance of MC_Instruction
   END_VAR
   // Ret_Val : No return value
BEGIN
   // Call of MC_Instruction
   #instMC(Axis := #axis);
END_FUNCTION

FUNCTION "LAnyAxis_UnpubHomeSyncAxis" : Void   // FC30060, SCL
TITLE = LAnyAxis_UnpubHomeSyncAxis
{ S7_Optimized_Access := 'TRUE' }
AUTHOR : tech.team.motioncontrol@siemens.com
FAMILY : AnyAxis
VERSION : 1.0
// Support: tech.team.motioncontrol@siemens.com
   VAR_INPUT
      axis : TO_SynchronousAxis;   // Axis specification
   END_VAR
   VAR_IN_OUT
      instMC : MC_HOME;   // Instance of MC_Instruction
   END_VAR
   // Ret_Val : No return value
BEGIN
   // Call of MC_Instruction
   #instMC(Axis := #axis);
END_FUNCTION

// folder: LAnyAxis_Blocks/InternalSubBlocks/MC_MoveAbsolute

FUNCTION "LAnyAxis_UnpubMoveAbsoluteSyncAxis" : Void   // FC30007, SCL
TITLE = LAnyAxis_UnpubMoveAbsoluteSyncAxis
{ S7_Optimized_Access := 'TRUE' }
AUTHOR : tech.team.motioncontrol@siemens.com
FAMILY : AnyAxis
VERSION : 1.0
// Support: tech.team.motioncontrol@siemens.com
   VAR_INPUT
      axis : TO_SynchronousAxis;   // Axis specification
   END_VAR
   VAR_IN_OUT
      instMC : MC_MOVEABSOLUTE;   // Instance of MC_Instruction
   END_VAR
   // Ret_Val : No return value
BEGIN
   // Call of MC_Instruction
   #instMC(Axis := #axis);
END_FUNCTION

// folder: LAnyAxis_Blocks/InternalSubBlocks/MC_MoveJog

